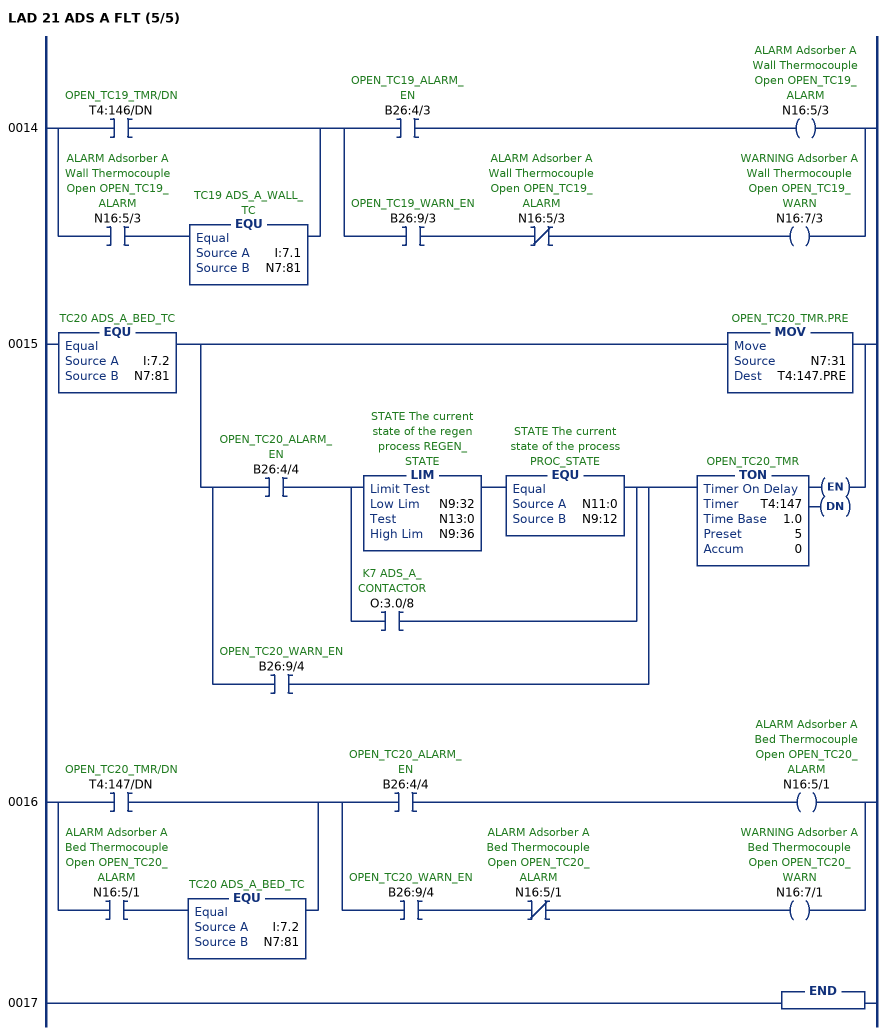
% Rung: 14 %
SOR BST XIC T4:146/DN NXB XIC N16:5/3 EQU I:7.1 N7:81 BND BST XIC B26:4/3 OTE N16:5/3 NXB XIC B26:9/3 XIO N16:5/3 OTE N16:7/3 BND EOR
%   T4:146  OPEN_TC19_TMR %
%   N16:5/3  OPEN_TC19_ALARM  "ALARM Adsorber A Wall Thermocouple Open" %
%   I:7.1  ADS_A_WALL_TC  "TC19" %
%   N7:81  TC_OPEN_SP  "CONFIG The value read by an open TC input" %
%   B26:4/3  OPEN_TC19_ALARM_EN %
%   B26:9/3  OPEN_TC19_WARN_EN %
%   N16:7/3  OPEN_TC19_WARN  "WARNING Adsorber A Wall Thermocouple Open" %
% Rung: 15 %
SOR EQU I:7.2 N7:81 BST MOV N7:31 T4:147.PRE NXB BST XIC B26:4/4 BST LIM N9:32 N13:0 N9:36 EQU N11:0 N9:12 NXB XIC O:3.0/8 BND NXB XIC B26:9/4 BND TON T4:147 1.0 5 0 BND EOR
%   I:7.2  ADS_A_BED_TC  "TC20" %
%   N7:81  TC_OPEN_SP  "CONFIG The value read by an open TC input" %
%   N7:31  OPEN_TC_DLY %
%   T4:147  OPEN_TC20_TMR %
%   B26:4/4  OPEN_TC20_ALARM_EN %
%   N9:32  REGEN_VENT  "STATE Regen Vent" %
%   N13:0  REGEN_STATE  "STATE The current state of the regen process" %
%   N9:36  REGEN_COOL  "STATE Regen Cool" %
%   N11:0  PROC_STATE  "STATE The current state of the process" %
%   N9:12  PROC_PFY_B_REG_A  "STATE Process Purify B" %
%   O:3.0/8  ADS_A_CONTACTOR  "K7" %
%   B26:9/4  OPEN_TC20_WARN_EN %
% Rung: 16 %
SOR BST XIC T4:147/DN NXB XIC N16:5/1 EQU I:7.2 N7:81 BND BST XIC B26:4/4 OTE N16:5/1 NXB XIC B26:9/4 XIO N16:5/1 OTE N16:7/1 BND EOR
%   T4:147  OPEN_TC20_TMR %
%   N16:5/1  OPEN_TC20_ALARM  "ALARM Adsorber A Bed Thermocouple Open" %
%   I:7.2  ADS_A_BED_TC  "TC20" %
%   N7:81  TC_OPEN_SP  "CONFIG The value read by an open TC input" %
%   B26:4/4  OPEN_TC20_ALARM_EN %
%   B26:9/4  OPEN_TC20_WARN_EN %
%   N16:7/1  OPEN_TC20_WARN  "WARNING Adsorber A Bed Thermocouple Open" %
% Rung: 17 %
SOR END EOR

LADDER 22 "ADS B"    % Controld Adsorber B %
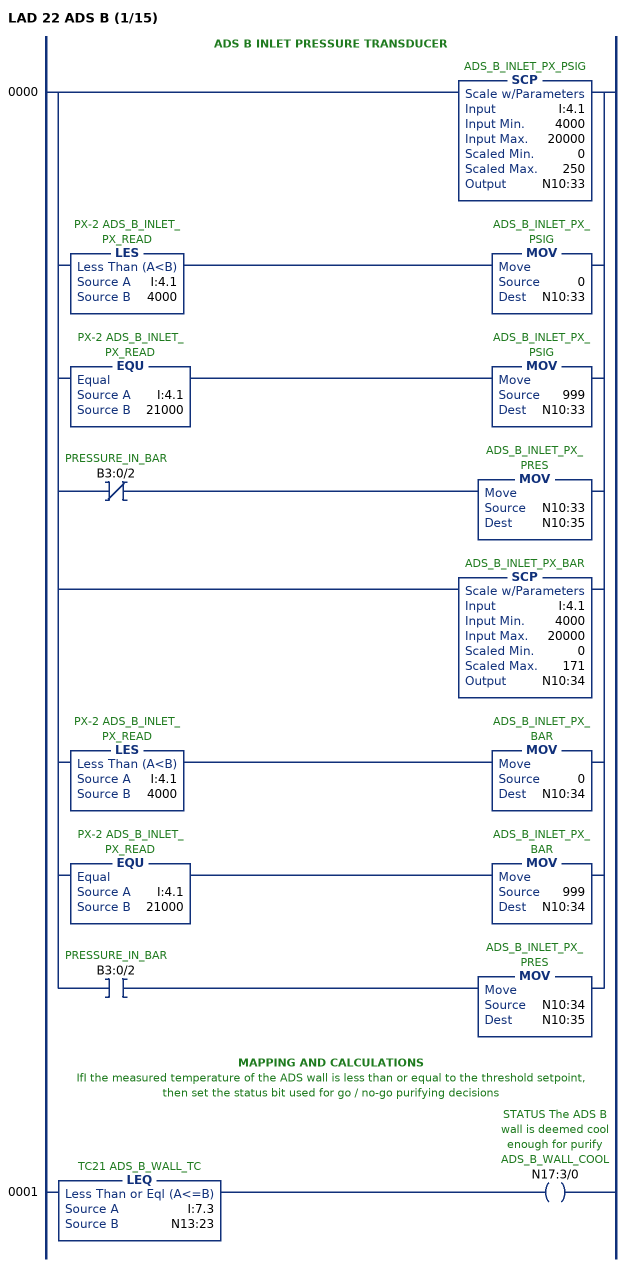
% Rung: 0 %
% TITLE: ADS B INLET PRESSURE TRANSDUCER %
SOR BST SCP I:4.1 4000 20000 0 250 N10:33 NXB LES I:4.1 4000 MOV 0 N10:33 NXB EQU I:4.1 21000 MOV 999 N10:33 NXB XIO B3:0/2 MOV N10:33 N10:35 NXB SCP I:4.1 4000 20000 0 171 N10:34 NXB LES I:4.1 4000 MOV 0 N10:34 NXB EQU I:4.1 21000 MOV 999 N10:34 NXB XIC B3:0/2 MOV N10:34 N10:35 BND EOR
%   I:4.1  ADS_B_INLET_PX_READ  "PX-2" %
%   N10:33  ADS_B_INLET_PX_PSIG %
%   B3:0/2  PRESSURE_IN_BAR %
%   N10:35  ADS_B_INLET_PX_PRES %
%   N10:34  ADS_B_INLET_PX_BAR %
% Rung: 1 %
% TITLE: MAPPING AND CALCULATIONS %
% IfI the measured temperature of the ADS wall is less than or equal to the threshold setpoint, then set the status bit used for go / no-go purifying decisions %
SOR LEQ I:7.3 N13:23 OTE N17:3/0 EOR
%   I:7.3  ADS_B_WALL_TC  "TC21" %
%   N13:23  ADS_WALL_TEMP_COOL  "CONFIG The temp at which the adsorber wall is deemed to be cool enough to purify" %
%   N17:3/0  ADS_B_WALL_COOL  "STATUS The ADS B wall is deemed cool enough for purify" %

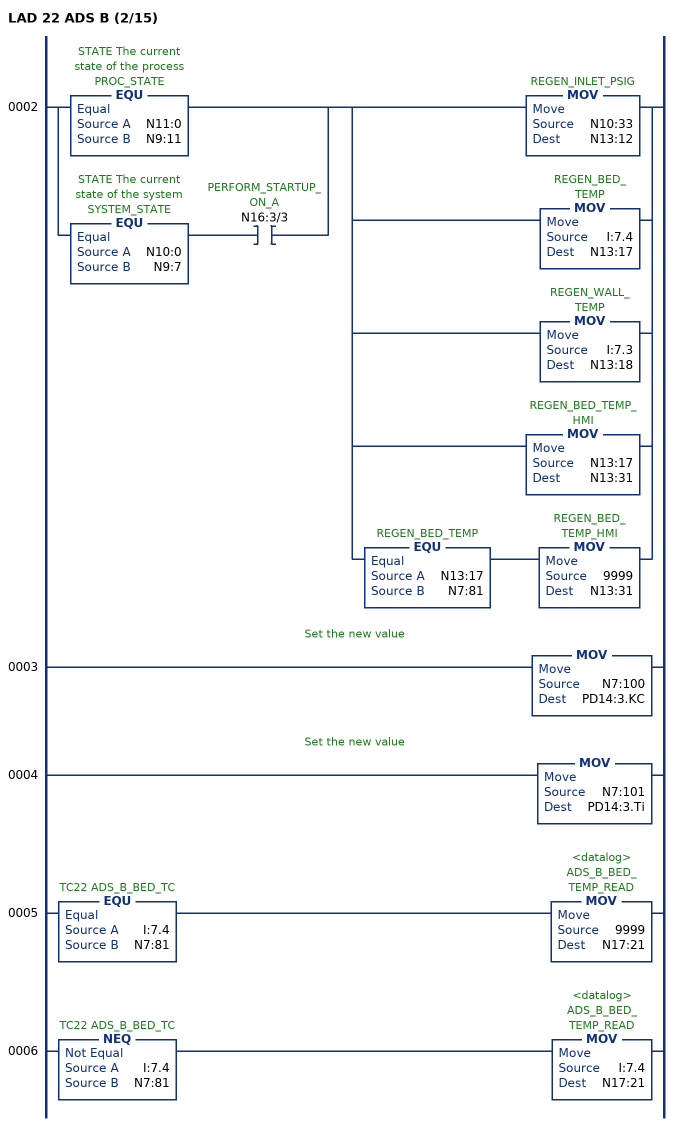
% Rung: 2 %
SOR BST EQU N11:0 N9:11 NXB EQU N10:0 N9:7 XIC N16:3/3 BND BST MOV N10:33 N13:12 NXB MOV I:7.4 N13:17 NXB MOV I:7.3 N13:18 NXB MOV N13:17 N13:31 NXB EQU N13:17 N7:81 MOV 9999 N13:31 BND EOR
%   N11:0  PROC_STATE  "STATE The current state of the process" %
%   N9:11  PROC_PFY_A_REG_B  "STATE Process Purify A" %
%   N10:0  SYSTEM_STATE  "STATE The current state of the system" %
%   N9:7  SYSTEM_COLD_START %
%   N16:3/3  PERFORM_STARTUP_ON_A %
%   N10:33  ADS_B_INLET_PX_PSIG %
%   N13:12  REGEN_INLET_PSIG %
%   I:7.4  ADS_B_BED_TC  "TC22" %
%   N13:17  REGEN_BED_TEMP %
%   I:7.3  ADS_B_WALL_TC  "TC21" %
%   N13:18  REGEN_WALL_TEMP %
%   N13:31  REGEN_BED_TEMP_HMI %
%   N7:81  TC_OPEN_SP  "CONFIG The value read by an open TC input" %
% Rung: 3 %
% Set the new value %
SOR MOV N7:100 PD14:3.KC EOR
%   N7:100  BLANKET_P  "CONFIG Blanket Proportional Gain New" %
% Rung: 4 %
% Set the new value %
SOR MOV N7:101 PD14:3.Ti EOR
%   N7:101  BLANKET_I  "CONFIG Blanket Integral Gain New" %
% Rung: 5 %
SOR EQU I:7.4 N7:81 MOV 9999 N17:21 EOR
%   I:7.4  ADS_B_BED_TC  "TC22" %
%   N7:81  TC_OPEN_SP  "CONFIG The value read by an open TC input" %
%   N17:21  ADS_B_BED_TEMP_READ  "<datalog>" %
% Rung: 6 %
SOR NEQ I:7.4 N7:81 MOV I:7.4 N17:21 EOR
%   I:7.4  ADS_B_BED_TC  "TC22" %
%   N7:81  TC_OPEN_SP  "CONFIG The value read by an open TC input" %
%   N17:21  ADS_B_BED_TEMP_READ  "<datalog>" %

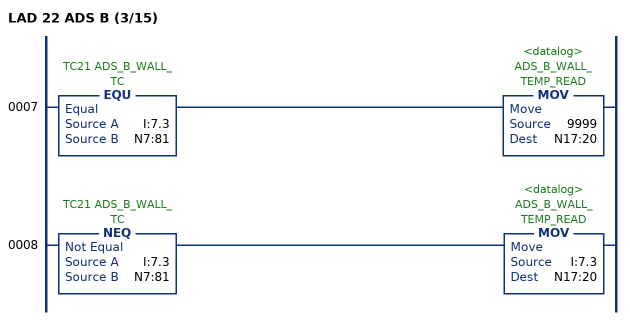
% Rung: 7 %
SOR EQU I:7.3 N7:81 MOV 9999 N17:20 EOR
%   I:7.3  ADS_B_WALL_TC  "TC21" %
%   N7:81  TC_OPEN_SP  "CONFIG The value read by an open TC input" %
%   N17:20  ADS_B_WALL_TEMP_READ  "<datalog>" %
% Rung: 8 %
SOR NEQ I:7.3 N7:81 MOV I:7.3 N17:20 EOR
%   I:7.3  ADS_B_WALL_TC  "TC21" %
%   N7:81  TC_OPEN_SP  "CONFIG The value read by an open TC input" %
%   N17:20  ADS_B_WALL_TEMP_READ  "<datalog>" %

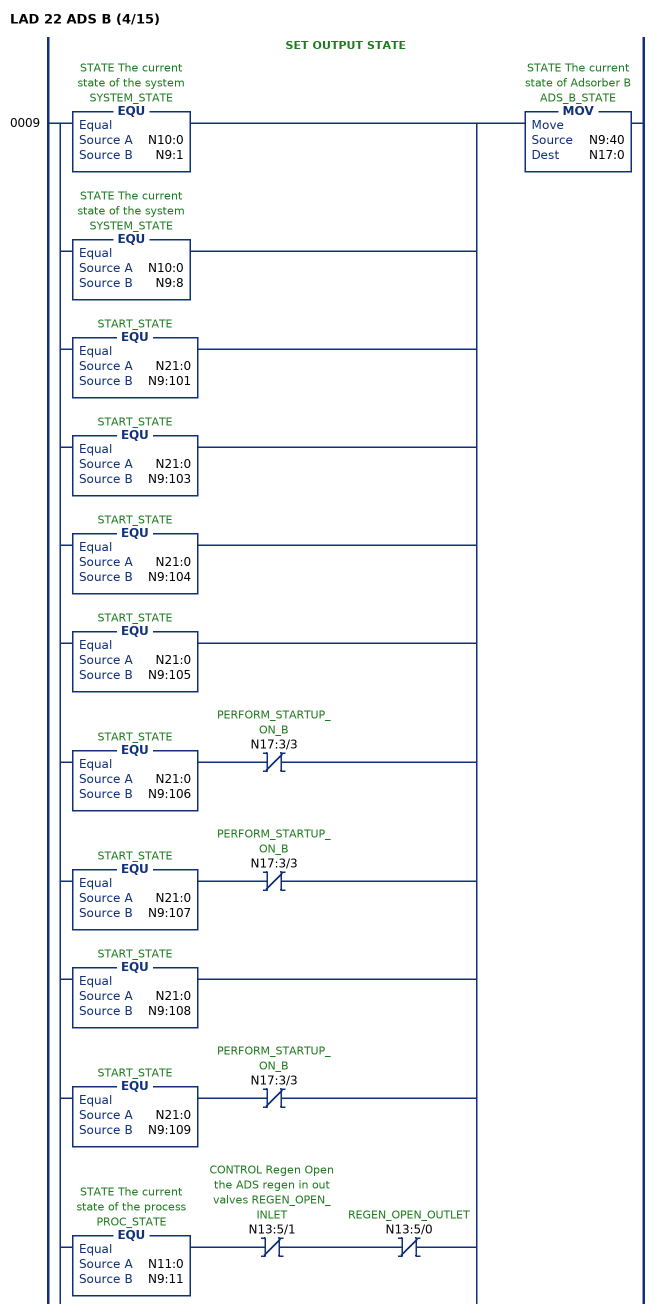

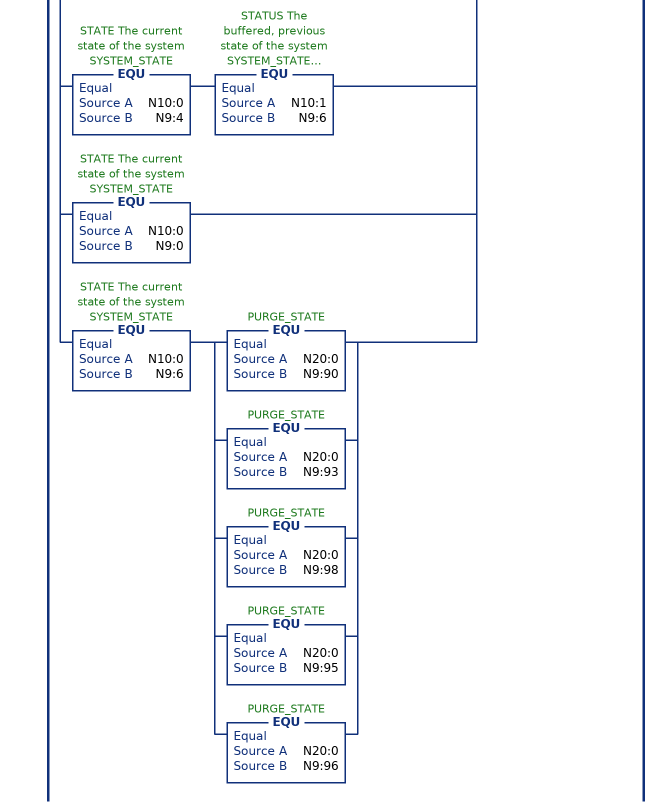
% Rung: 9 %
% TITLE: SET OUTPUT STATE %
SOR BST EQU N10:0 N9:1 NXB EQU N10:0 N9:8 NXB BST EQU N21:0 N9:101 NXB EQU N21:0 N9:103 NXB EQU N21:0 N9:104 NXB EQU N21:0 N9:105 NXB EQU N21:0 N9:106 XIO N17:3/3 NXB EQU N21:0 N9:107 XIO N17:3/3 NXB EQU N21:0 N9:108 NXB EQU N21:0 N9:109 XIO N17:3/3 BND NXB EQU N11:0 N9:11 XIO N13:5/1 XIO N13:5/0 NXB EQU N10:0 N9:4 EQU N10:1 N9:6 NXB EQU N10:0 N9:0 NXB EQU N10:0 N9:6 BST EQU N20:0 N9:90 NXB EQU N20:0 N9:93 NXB EQU N20:0 N9:98 NXB EQU N20:0 N9:95 NXB EQU N20:0 N9:96 BND BND MOV N9:40 N17:0 EOR
%   N10:0  SYSTEM_STATE  "STATE The current state of the system" %
%   N9:1  SYSTEM_STANDBY  "STATE System Process" %
%   N9:8  SYSTEM_SUPPLEMENTAL %
%   N21:0  START_STATE %
%   N9:101  START_COOL %
%   N9:103  START_VENT_GET_1 %
%   N9:104  START_HEAT %
%   N9:105  START_VENT_ALL %
%   N9:106  START_BACKFILL_1 %
%   N17:3/3  PERFORM_STARTUP_ON_B %
%   N9:107  START_VENT_ADS_2 %
%   N9:108  START_VENT_GET_2 %
%   N9:109  START_BACKFILL_2 %
%   N11:0  PROC_STATE  "STATE The current state of the process" %
%   N9:11  PROC_PFY_A_REG_B  "STATE Process Purify A" %
%   N13:5/1  REGEN_OPEN_INLET  "CONTROL Regen Open the ADS regen in out valves" %
%   N13:5/0  REGEN_OPEN_OUTLET %
%   N9:4  SYSTEM_ALARM  "STATE System Alarm" %
%   N10:1  SYSTEM_STATE_BUFFER  "STATUS The buffered, previous state of the system" %
%   N9:6  SYSTEM_PURGE %
%   N9:0  SYSTEM_OFFLINE %
%   N20:0  PURGE_STATE %
%   N9:90  PURGE_IDLE %
%   N9:93  PURGE_VENT_GETTER %
%   N9:98  PURGE_VENT_GET_2 %
%   N9:95  PURGE_FINAL_VENT %
%   N9:96  PURGE_DONE %
%   N9:40  ADS_STANDBY  "STATE ADS Standby" %
%   N17:0  ADS_B_STATE  "STATE The current state of Adsorber B" %

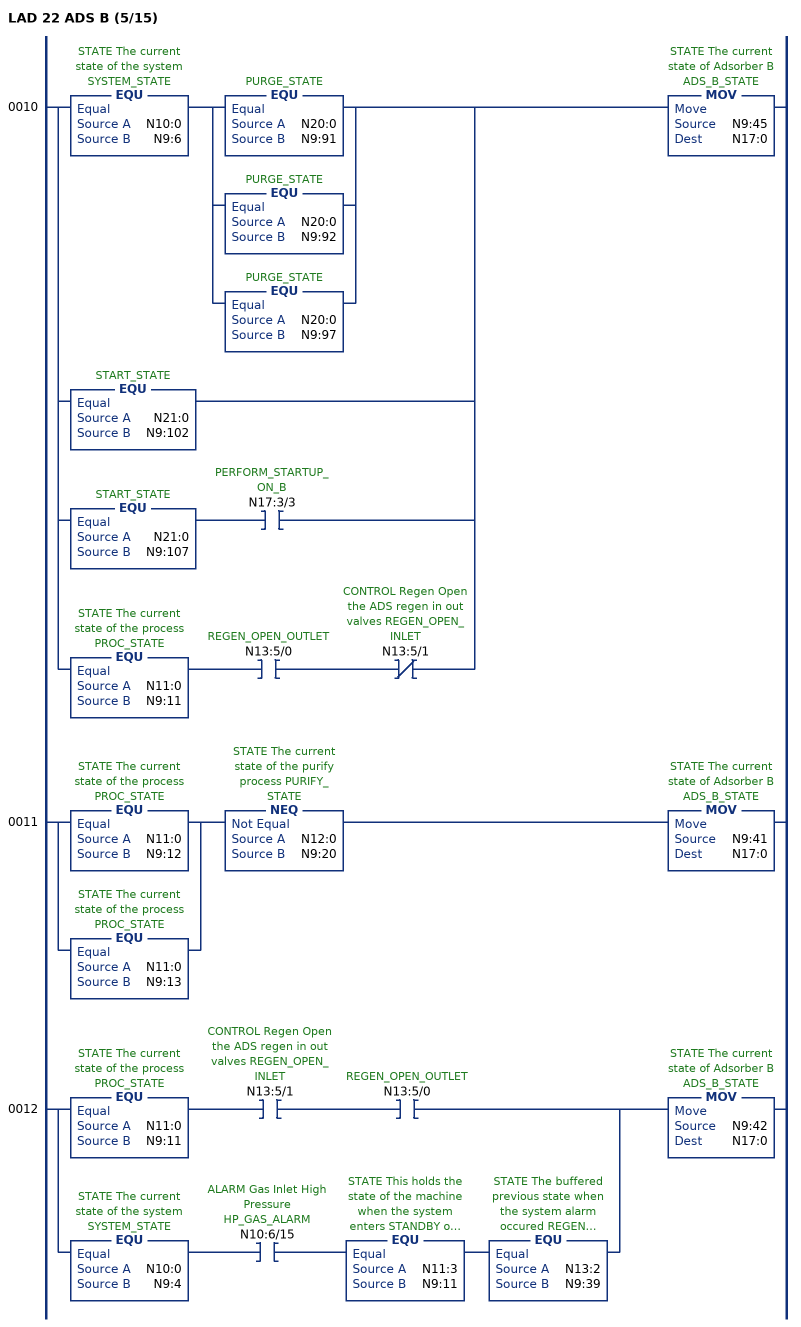
% Rung: 10 %
SOR BST EQU N10:0 N9:6 BST EQU N20:0 N9:91 NXB EQU N20:0 N9:92 NXB EQU N20:0 N9:97 BND NXB BST EQU N21:0 N9:102 NXB EQU N21:0 N9:107 XIC N17:3/3 BND NXB EQU N11:0 N9:11 XIC N13:5/0 XIO N13:5/1 BND MOV N9:45 N17:0 EOR
%   N10:0  SYSTEM_STATE  "STATE The current state of the system" %
%   N9:6  SYSTEM_PURGE %
%   N20:0  PURGE_STATE %
%   N9:91  PURGE_INIT_VENT %
%   N9:92  PURGE_VENT_ADSORBER %
%   N9:97  PURGE_VENT_ADS_2 %
%   N21:0  START_STATE %
%   N9:102  START_VENT_ADS_1 %
%   N9:107  START_VENT_ADS_2 %
%   N17:3/3  PERFORM_STARTUP_ON_B %
%   N11:0  PROC_STATE  "STATE The current state of the process" %
%   N9:11  PROC_PFY_A_REG_B  "STATE Process Purify A" %
%   N13:5/0  REGEN_OPEN_OUTLET %
%   N13:5/1  REGEN_OPEN_INLET  "CONTROL Regen Open the ADS regen in out valves" %
%   N9:45  ADS_VENT %
%   N17:0  ADS_B_STATE  "STATE The current state of Adsorber B" %
% Rung: 11 %
SOR BST EQU N11:0 N9:12 NXB EQU N11:0 N9:13 BND NEQ N12:0 N9:20 MOV N9:41 N17:0 EOR
%   N11:0  PROC_STATE  "STATE The current state of the process" %
%   N9:12  PROC_PFY_B_REG_A  "STATE Process Purify B" %
%   N9:13  PROC_OVERLAP  "STATE Process Purify Overlap" %
%   N12:0  PURIFY_STATE  "STATE The current state of the purify process" %
%   N9:20  PURIFY_STANDBY  "STATE Purify Standby" %
%   N9:41  ADS_PURIFY  "STATE ADS Purify" %
%   N17:0  ADS_B_STATE  "STATE The current state of Adsorber B" %
% Rung: 12 %
SOR BST EQU N11:0 N9:11 XIC N13:5/1 XIC N13:5/0 NXB EQU N10:0 N9:4 XIC N10:6/15 EQU N11:3 N9:11 EQU N13:2 N9:39 BND MOV N9:42 N17:0 EOR
%   N11:0  PROC_STATE  "STATE The current state of the process" %
%   N9:11  PROC_PFY_A_REG_B  "STATE Process Purify A" %
%   N13:5/1  REGEN_OPEN_INLET  "CONTROL Regen Open the ADS regen in out valves" %
%   N13:5/0  REGEN_OPEN_OUTLET %
%   N10:0  SYSTEM_STATE  "STATE The current state of the system" %
%   N9:4  SYSTEM_ALARM  "STATE System Alarm" %
%   N10:6/15  HP_GAS_ALARM  "ALARM Gas Inlet High Pressure" %
%   N11:3  PROC_STATE_BUFFER  "STATE This holds the state of the machine when the system enters STANDBY or ALARM" %
%   N13:2  REGEN_SYSTEM_BUFFER  "STATE The buffered previous state when the system alarm occured" %
%   N9:39  REGEN_BACKFILL %
%   N9:42  ADS_REGEN  "STATE ADS Regen" %
%   N17:0  ADS_B_STATE  "STATE The current state of Adsorber B" %

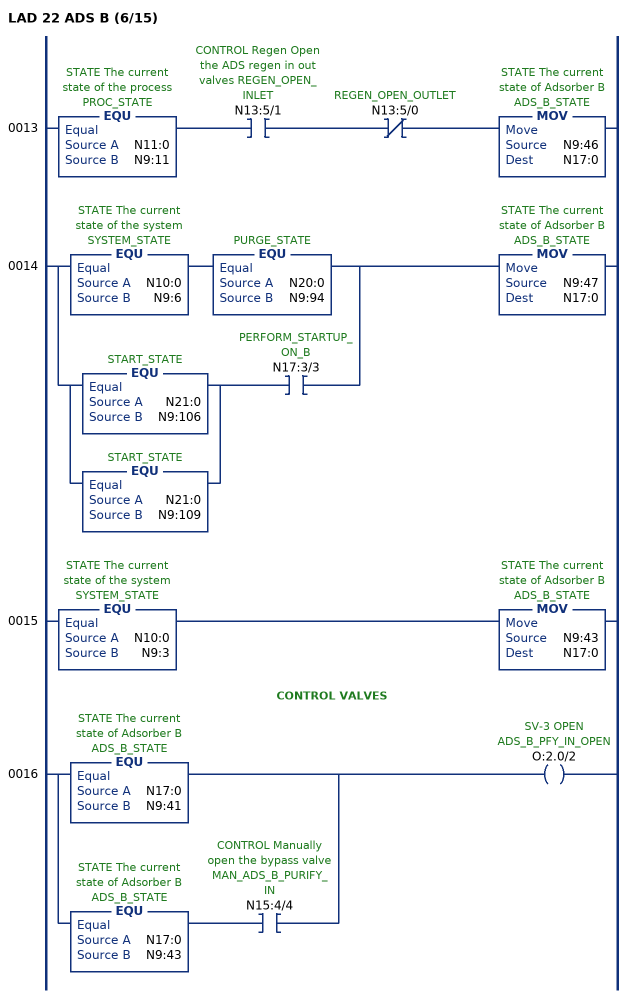
% Rung: 13 %
SOR EQU N11:0 N9:11 XIC N13:5/1 XIO N13:5/0 MOV N9:46 N17:0 EOR
%   N11:0  PROC_STATE  "STATE The current state of the process" %
%   N9:11  PROC_PFY_A_REG_B  "STATE Process Purify A" %
%   N13:5/1  REGEN_OPEN_INLET  "CONTROL Regen Open the ADS regen in out valves" %
%   N13:5/0  REGEN_OPEN_OUTLET %
%   N9:46  ADS_REGEN_BACKFILL %
%   N17:0  ADS_B_STATE  "STATE The current state of Adsorber B" %
% Rung: 14 %
SOR BST EQU N10:0 N9:6 EQU N20:0 N9:94 NXB BST EQU N21:0 N9:106 NXB EQU N21:0 N9:109 BND XIC N17:3/3 BND MOV N9:47 N17:0 EOR
%   N10:0  SYSTEM_STATE  "STATE The current state of the system" %
%   N9:6  SYSTEM_PURGE %
%   N20:0  PURGE_STATE %
%   N9:94  PURGE_BACKFILL %
%   N21:0  START_STATE %
%   N9:106  START_BACKFILL_1 %
%   N9:109  START_BACKFILL_2 %
%   N17:3/3  PERFORM_STARTUP_ON_B %
%   N9:47  ADS_BACKFILL %
%   N17:0  ADS_B_STATE  "STATE The current state of Adsorber B" %
% Rung: 15 %
SOR EQU N10:0 N9:3 MOV N9:43 N17:0 EOR
%   N10:0  SYSTEM_STATE  "STATE The current state of the system" %
%   N9:3  SYSTEM_MANUAL  "STATE System Manual" %
%   N9:43  ADS_MANUAL  "STATE ADS Manual" %
%   N17:0  ADS_B_STATE  "STATE The current state of Adsorber B" %
% Rung: 16 %
% TITLE: CONTROL VALVES %
SOR BST EQU N17:0 N9:41 NXB EQU N17:0 N9:43 XIC N15:4/4 BND OTE O:2.0/2 EOR
%   N17:0  ADS_B_STATE  "STATE The current state of Adsorber B" %
%   N9:41  ADS_PURIFY  "STATE ADS Purify" %
%   N9:43  ADS_MANUAL  "STATE ADS Manual" %
%   N15:4/4  MAN_ADS_B_PURIFY_IN  "CONTROL Manually open the bypass valve" %
%   O:2.0/2  ADS_B_PFY_IN_OPEN  "SV-3 OPEN" %

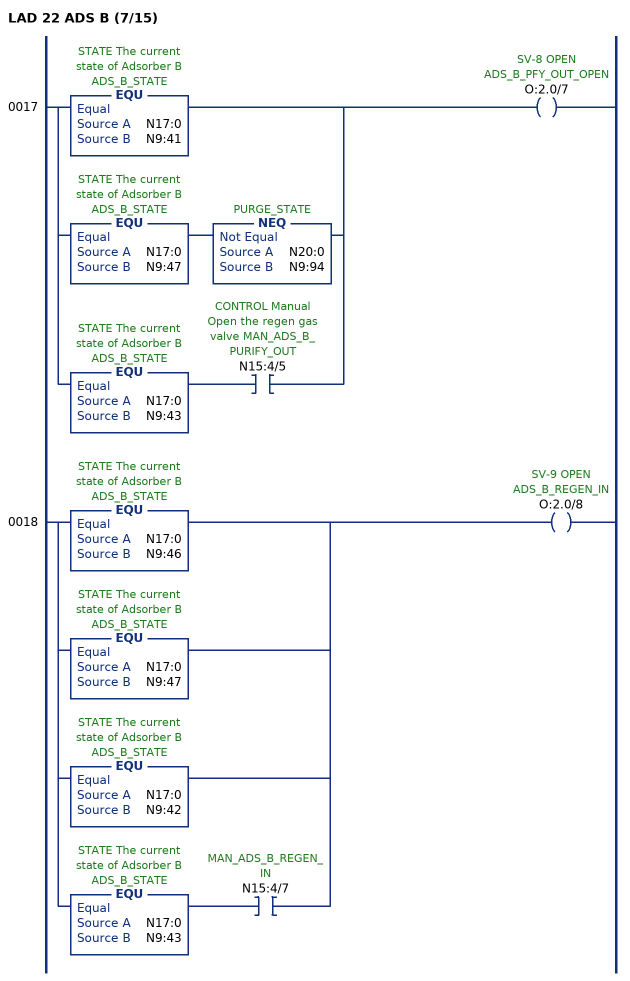
% Rung: 17 %
SOR BST EQU N17:0 N9:41 NXB EQU N17:0 N9:47 NEQ N20:0 N9:94 NXB EQU N17:0 N9:43 XIC N15:4/5 BND OTE O:2.0/7 EOR
%   N17:0  ADS_B_STATE  "STATE The current state of Adsorber B" %
%   N9:41  ADS_PURIFY  "STATE ADS Purify" %
%   N9:47  ADS_BACKFILL %
%   N20:0  PURGE_STATE %
%   N9:94  PURGE_BACKFILL %
%   N9:43  ADS_MANUAL  "STATE ADS Manual" %
%   N15:4/5  MAN_ADS_B_PURIFY_OUT  "CONTROL Manual Open the regen gas valve" %
%   O:2.0/7  ADS_B_PFY_OUT_OPEN  "SV-8 OPEN" %
% Rung: 18 %
SOR BST EQU N17:0 N9:46 NXB EQU N17:0 N9:47 NXB EQU N17:0 N9:42 NXB EQU N17:0 N9:43 XIC N15:4/7 BND OTE O:2.0/8 EOR
%   N17:0  ADS_B_STATE  "STATE The current state of Adsorber B" %
%   N9:46  ADS_REGEN_BACKFILL %
%   N9:47  ADS_BACKFILL %
%   N9:42  ADS_REGEN  "STATE ADS Regen" %
%   N9:43  ADS_MANUAL  "STATE ADS Manual" %
%   N15:4/7  MAN_ADS_B_REGEN_IN %
%   O:2.0/8  ADS_B_REGEN_IN  "SV-9 OPEN" %

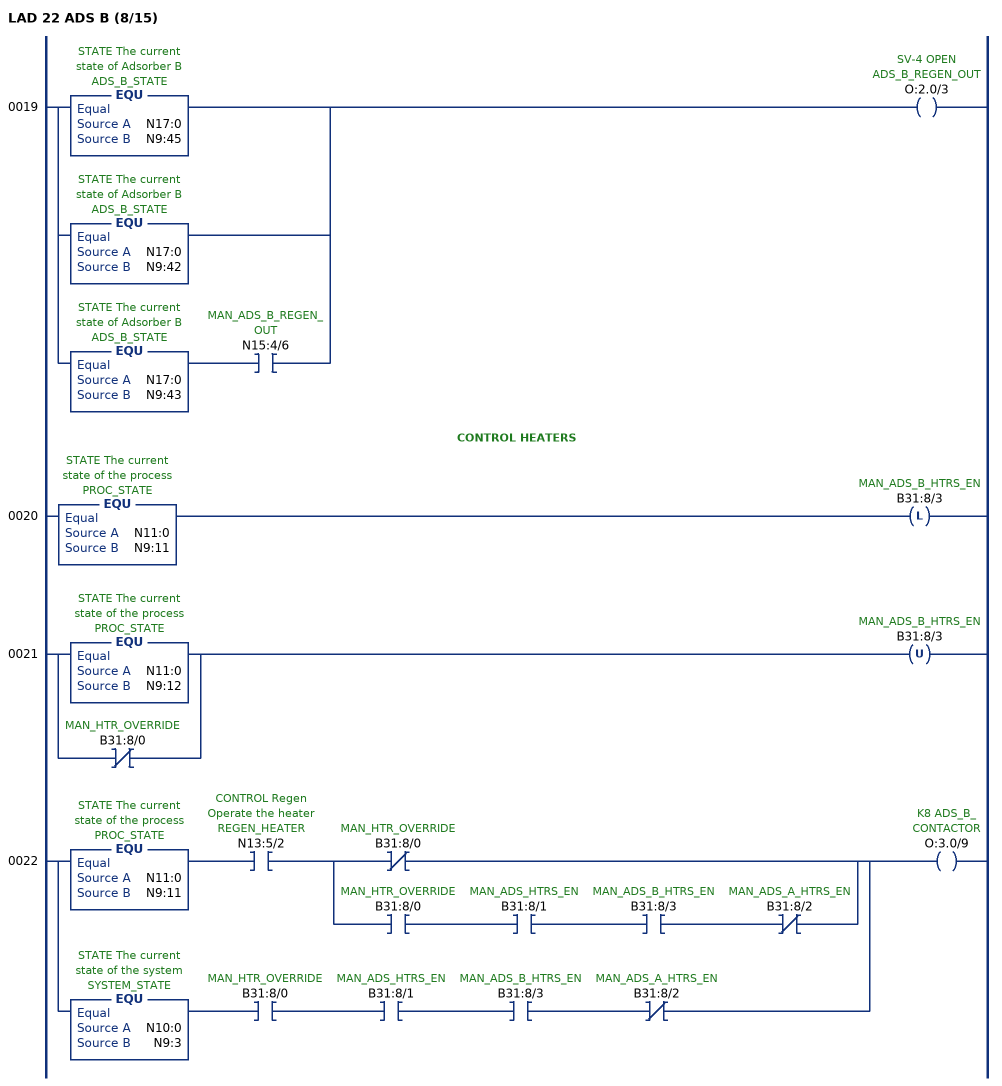
% Rung: 19 %
SOR BST EQU N17:0 N9:45 NXB EQU N17:0 N9:42 NXB EQU N17:0 N9:43 XIC N15:4/6 BND OTE O:2.0/3 EOR
%   N17:0  ADS_B_STATE  "STATE The current state of Adsorber B" %
%   N9:45  ADS_VENT %
%   N9:42  ADS_REGEN  "STATE ADS Regen" %
%   N9:43  ADS_MANUAL  "STATE ADS Manual" %
%   N15:4/6  MAN_ADS_B_REGEN_OUT %
%   O:2.0/3  ADS_B_REGEN_OUT  "SV-4 OPEN" %
% Rung: 20 %
% TITLE: CONTROL HEATERS %
SOR EQU N11:0 N9:11 OTL B31:8/3 EOR
%   N11:0  PROC_STATE  "STATE The current state of the process" %
%   N9:11  PROC_PFY_A_REG_B  "STATE Process Purify A" %
%   B31:8/3  MAN_ADS_B_HTRS_EN %
% Rung: 21 %
SOR BST EQU N11:0 N9:12 NXB XIO B31:8/0 BND OTU B31:8/3 EOR
%   N11:0  PROC_STATE  "STATE The current state of the process" %
%   N9:12  PROC_PFY_B_REG_A  "STATE Process Purify B" %
%   B31:8/0  MAN_HTR_OVERRIDE %
%   B31:8/3  MAN_ADS_B_HTRS_EN %
% Rung: 22 %
SOR BST EQU N11:0 N9:11 XIC N13:5/2 BST XIO B31:8/0 NXB XIC B31:8/0 XIC B31:8/1 XIC B31:8/3 XIO B31:8/2 BND NXB EQU N10:0 N9:3 XIC B31:8/0 XIC B31:8/1 XIC B31:8/3 XIO B31:8/2 BND OTE O:3.0/9 EOR
%   N11:0  PROC_STATE  "STATE The current state of the process" %
%   N9:11  PROC_PFY_A_REG_B  "STATE Process Purify A" %
%   N13:5/2  REGEN_HEATER  "CONTROL Regen Operate the heater" %
%   B31:8/0  MAN_HTR_OVERRIDE %
%   B31:8/1  MAN_ADS_HTRS_EN %
%   B31:8/3  MAN_ADS_B_HTRS_EN %
%   B31:8/2  MAN_ADS_A_HTRS_EN %
%   N10:0  SYSTEM_STATE  "STATE The current state of the system" %
%   N9:3  SYSTEM_MANUAL  "STATE System Manual" %
%   O:3.0/9  ADS_B_CONTACTOR  "K8" %

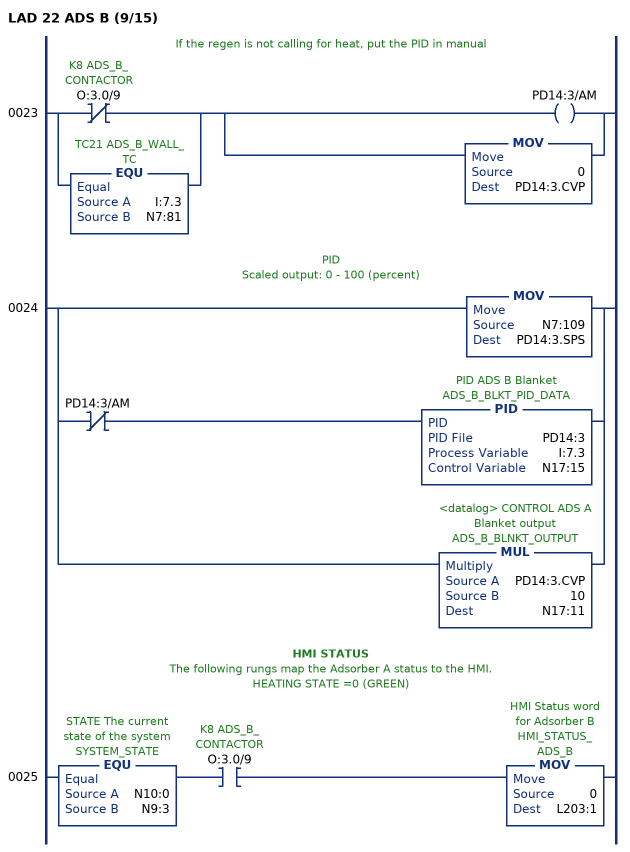
% Rung: 23 %
% If the regen is not calling for heat, put the PID in manual %
SOR BST XIO O:3.0/9 NXB EQU I:7.3 N7:81 BND BST OTE PD14:3/AM NXB MOV 0 PD14:3.CVP BND EOR
%   O:3.0/9  ADS_B_CONTACTOR  "K8" %
%   I:7.3  ADS_B_WALL_TC  "TC21" %
%   N7:81  TC_OPEN_SP  "CONFIG The value read by an open TC input" %
% Rung: 24 %
% PID
% Scaled output: 0 - 100 (percent) %
SOR BST MOV N7:109 PD14:3.SPS NXB XIO PD14:3/AM PID PD14:3 I:7.3 N17:15 NXB MUL PD14:3.CVP 10 N17:11 BND EOR
%   N7:109  BLANKET_SP  "<datalog> CONTROL Blanket PID Setpoint" %
%   PD14:3  ADS_B_BLKT_PID_DATA  "PID ADS B Blanket" %
%   I:7.3  ADS_B_WALL_TC  "TC21" %
%   N17:15  ADS_B_BLKT_OUTPT_RAW  "CONTROL ADS B Blanket PID Output Raw" %
%   N17:11  ADS_B_BLNKT_OUTPUT  "<datalog> CONTROL ADS A Blanket output" %
% Rung: 25 %
% TITLE: HMI STATUS %
% The following rungs map the Adsorber A status to the HMI.
% HEATING STATE =0 (GREEN) %
SOR EQU N10:0 N9:3 XIC O:3.0/9 MOV 0 L203:1 EOR
%   N10:0  SYSTEM_STATE  "STATE The current state of the system" %
%   N9:3  SYSTEM_MANUAL  "STATE System Manual" %
%   O:3.0/9  ADS_B_CONTACTOR  "K8" %
%   L203:1  HMI_STATUS_ADS_B  "HMI Status word for Adsorber B" %

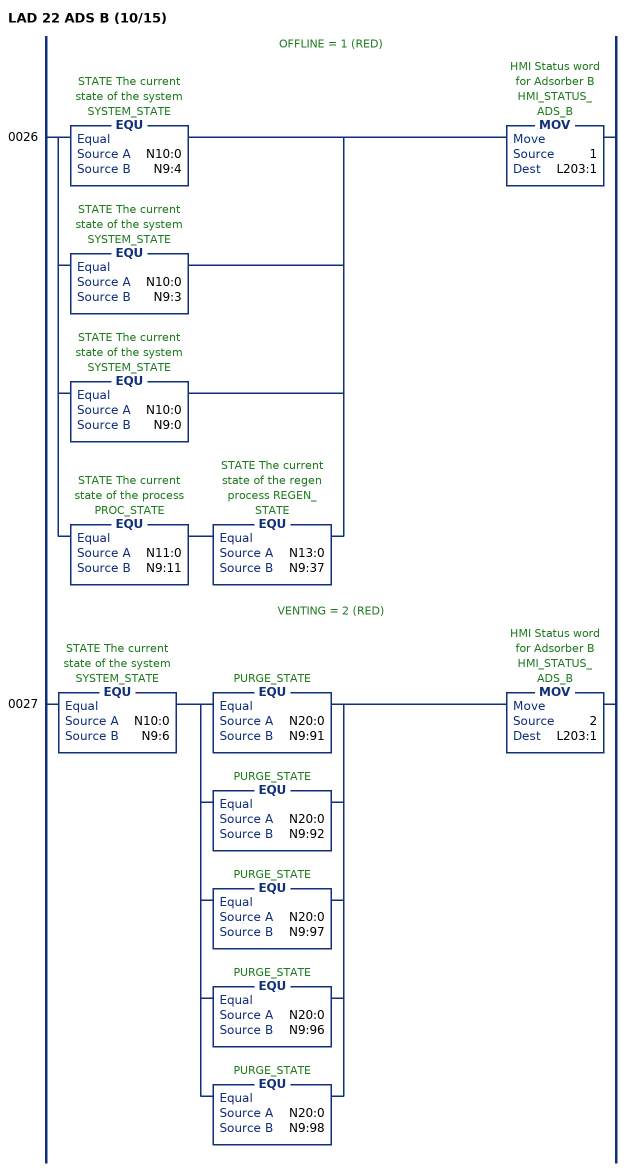
% Rung: 26 %
% OFFLINE = 1 (RED) %
SOR BST BST EQU N10:0 N9:4 NXB EQU N10:0 N9:3 NXB EQU N10:0 N9:0 BND NXB EQU N11:0 N9:11 EQU N13:0 N9:37 BND MOV 1 L203:1 EOR
%   N10:0  SYSTEM_STATE  "STATE The current state of the system" %
%   N9:4  SYSTEM_ALARM  "STATE System Alarm" %
%   N9:3  SYSTEM_MANUAL  "STATE System Manual" %
%   N9:0  SYSTEM_OFFLINE %
%   N11:0  PROC_STATE  "STATE The current state of the process" %
%   N9:11  PROC_PFY_A_REG_B  "STATE Process Purify A" %
%   N13:0  REGEN_STATE  "STATE The current state of the regen process" %
%   N9:37  REGEN_ALARM  "STATE Regen Alarm" %
%   L203:1  HMI_STATUS_ADS_B  "HMI Status word for Adsorber B" %
% Rung: 27 %
% VENTING = 2 (RED) %
SOR EQU N10:0 N9:6 BST EQU N20:0 N9:91 NXB EQU N20:0 N9:92 NXB EQU N20:0 N9:97 NXB EQU N20:0 N9:96 NXB EQU N20:0 N9:98 BND MOV 2 L203:1 EOR
%   N10:0  SYSTEM_STATE  "STATE The current state of the system" %
%   N9:6  SYSTEM_PURGE %
%   N20:0  PURGE_STATE %
%   N9:91  PURGE_INIT_VENT %
%   N9:92  PURGE_VENT_ADSORBER %
%   N9:97  PURGE_VENT_ADS_2 %
%   N9:96  PURGE_DONE %
%   N9:98  PURGE_VENT_GET_2 %
%   L203:1  HMI_STATUS_ADS_B  "HMI Status word for Adsorber B" %

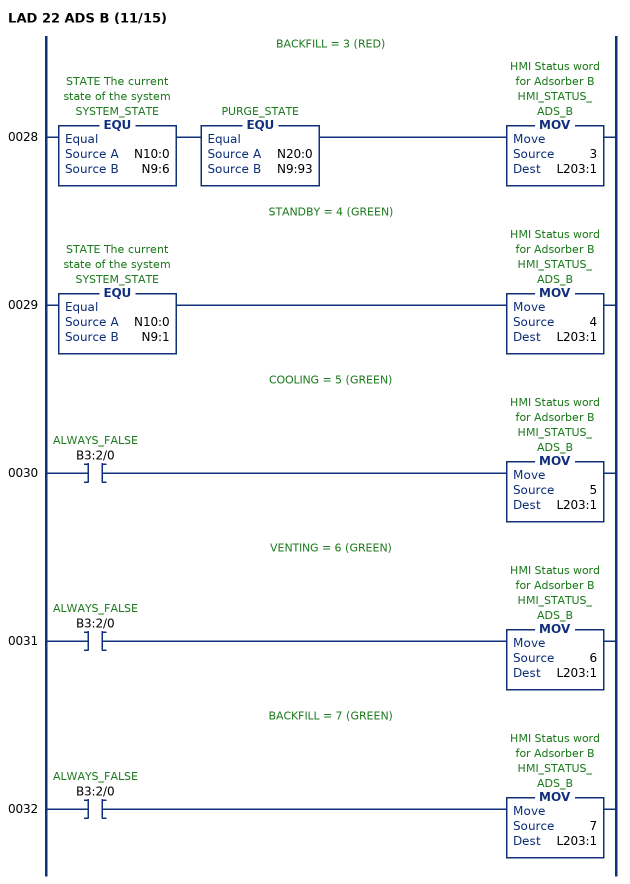
% Rung: 28 %
% BACKFILL = 3 (RED) %
SOR EQU N10:0 N9:6 EQU N20:0 N9:93 MOV 3 L203:1 EOR
%   N10:0  SYSTEM_STATE  "STATE The current state of the system" %
%   N9:6  SYSTEM_PURGE %
%   N20:0  PURGE_STATE %
%   N9:93  PURGE_VENT_GETTER %
%   L203:1  HMI_STATUS_ADS_B  "HMI Status word for Adsorber B" %
% Rung: 29 %
% STANDBY = 4 (GREEN) %
SOR EQU N10:0 N9:1 MOV 4 L203:1 EOR
%   N10:0  SYSTEM_STATE  "STATE The current state of the system" %
%   N9:1  SYSTEM_STANDBY  "STATE System Process" %
%   L203:1  HMI_STATUS_ADS_B  "HMI Status word for Adsorber B" %
% Rung: 30 %
% COOLING = 5 (GREEN) %
SOR XIC B3:2/0 MOV 5 L203:1 EOR
%   B3:2/0  ALWAYS_FALSE %
%   L203:1  HMI_STATUS_ADS_B  "HMI Status word for Adsorber B" %
% Rung: 31 %
% VENTING = 6 (GREEN) %
SOR XIC B3:2/0 MOV 6 L203:1 EOR
%   B3:2/0  ALWAYS_FALSE %
%   L203:1  HMI_STATUS_ADS_B  "HMI Status word for Adsorber B" %
% Rung: 32 %
% BACKFILL = 7 (GREEN) %
SOR XIC B3:2/0 MOV 7 L203:1 EOR
%   B3:2/0  ALWAYS_FALSE %
%   L203:1  HMI_STATUS_ADS_B  "HMI Status word for Adsorber B" %

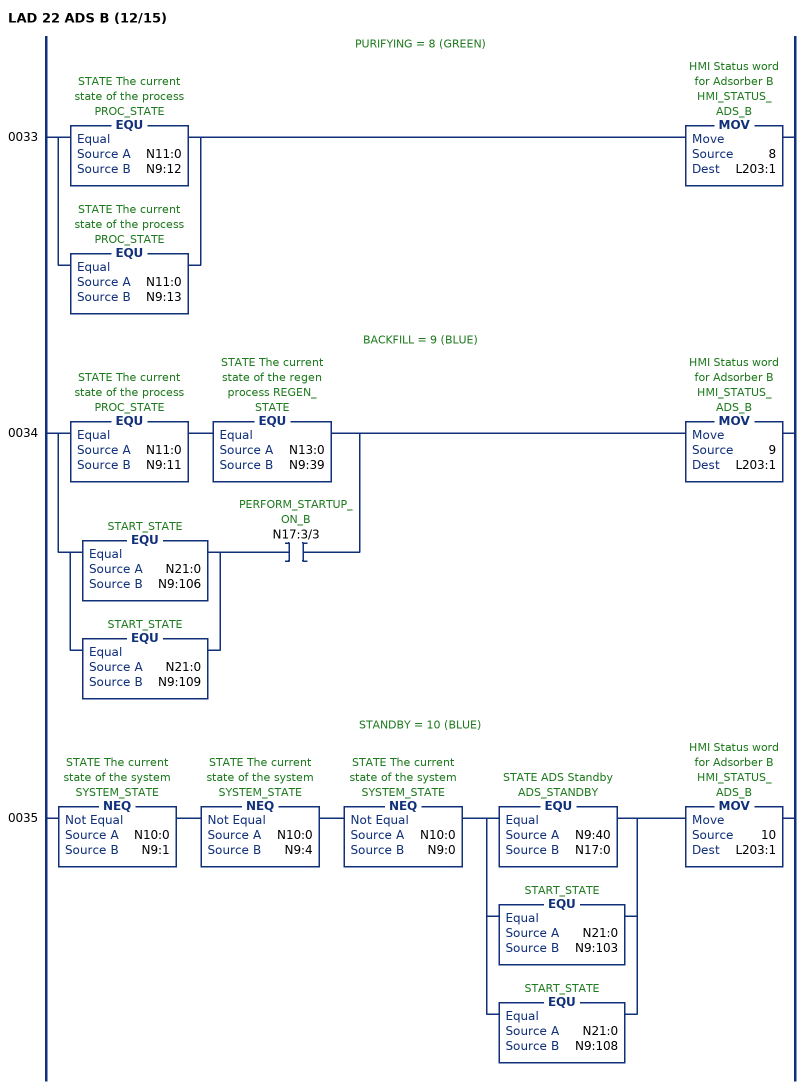
% Rung: 33 %
% PURIFYING = 8 (GREEN) %
SOR BST EQU N11:0 N9:12 NXB EQU N11:0 N9:13 BND MOV 8 L203:1 EOR
%   N11:0  PROC_STATE  "STATE The current state of the process" %
%   N9:12  PROC_PFY_B_REG_A  "STATE Process Purify B" %
%   N9:13  PROC_OVERLAP  "STATE Process Purify Overlap" %
%   L203:1  HMI_STATUS_ADS_B  "HMI Status word for Adsorber B" %
% Rung: 34 %
% BACKFILL = 9 (BLUE) %
SOR BST EQU N11:0 N9:11 EQU N13:0 N9:39 NXB BST EQU N21:0 N9:106 NXB EQU N21:0 N9:109 BND XIC N17:3/3 BND MOV 9 L203:1 EOR
%   N11:0  PROC_STATE  "STATE The current state of the process" %
%   N9:11  PROC_PFY_A_REG_B  "STATE Process Purify A" %
%   N13:0  REGEN_STATE  "STATE The current state of the regen process" %
%   N9:39  REGEN_BACKFILL %
%   N21:0  START_STATE %
%   N9:106  START_BACKFILL_1 %
%   N9:109  START_BACKFILL_2 %
%   N17:3/3  PERFORM_STARTUP_ON_B %
%   L203:1  HMI_STATUS_ADS_B  "HMI Status word for Adsorber B" %
% Rung: 35 %
% STANDBY = 10 (BLUE) %
SOR NEQ N10:0 N9:1 NEQ N10:0 N9:4 NEQ N10:0 N9:0 BST EQU N9:40 N17:0 NXB EQU N21:0 N9:103 NXB EQU N21:0 N9:108 BND MOV 10 L203:1 EOR
%   N10:0  SYSTEM_STATE  "STATE The current state of the system" %
%   N9:1  SYSTEM_STANDBY  "STATE System Process" %
%   N9:4  SYSTEM_ALARM  "STATE System Alarm" %
%   N9:0  SYSTEM_OFFLINE %
%   N9:40  ADS_STANDBY  "STATE ADS Standby" %
%   N17:0  ADS_B_STATE  "STATE The current state of Adsorber B" %
%   N21:0  START_STATE %
%   N9:103  START_VENT_GET_1 %
%   N9:108  START_VENT_GET_2 %
%   L203:1  HMI_STATUS_ADS_B  "HMI Status word for Adsorber B" %

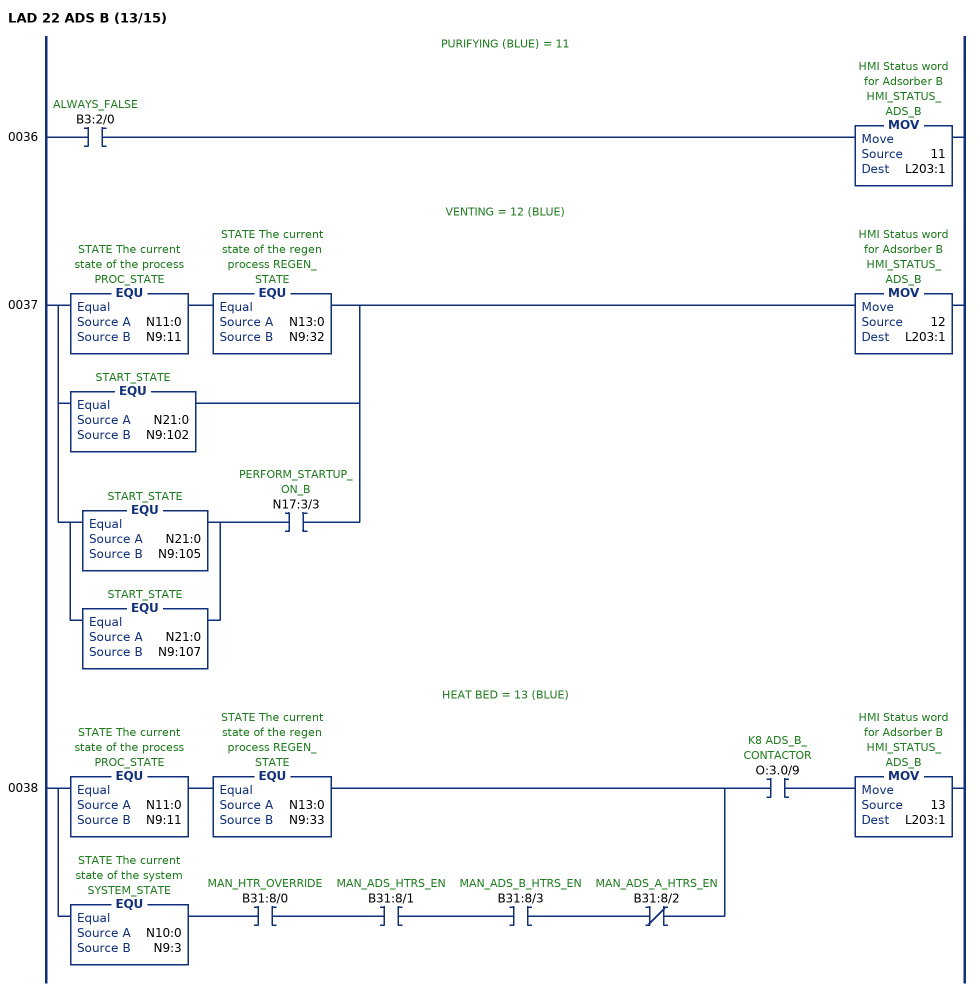
% Rung: 36 %
% PURIFYING (BLUE) = 11 %
SOR XIC B3:2/0 MOV 11 L203:1 EOR
%   B3:2/0  ALWAYS_FALSE %
%   L203:1  HMI_STATUS_ADS_B  "HMI Status word for Adsorber B" %
% Rung: 37 %
% VENTING = 12 (BLUE) %
SOR BST EQU N11:0 N9:11 EQU N13:0 N9:32 NXB BST EQU N21:0 N9:102 NXB BST EQU N21:0 N9:105 NXB EQU N21:0 N9:107 BND XIC N17:3/3 BND BND MOV 12 L203:1 EOR
%   N11:0  PROC_STATE  "STATE The current state of the process" %
%   N9:11  PROC_PFY_A_REG_B  "STATE Process Purify A" %
%   N13:0  REGEN_STATE  "STATE The current state of the regen process" %
%   N9:32  REGEN_VENT  "STATE Regen Vent" %
%   N21:0  START_STATE %
%   N9:102  START_VENT_ADS_1 %
%   N9:105  START_VENT_ALL %
%   N9:107  START_VENT_ADS_2 %
%   N17:3/3  PERFORM_STARTUP_ON_B %
%   L203:1  HMI_STATUS_ADS_B  "HMI Status word for Adsorber B" %
% Rung: 38 %
% HEAT BED = 13 (BLUE) %
SOR BST EQU N11:0 N9:11 EQU N13:0 N9:33 NXB EQU N10:0 N9:3 XIC B31:8/0 XIC B31:8/1 XIC B31:8/3 XIO B31:8/2 BND XIC O:3.0/9 MOV 13 L203:1 EOR
%   N11:0  PROC_STATE  "STATE The current state of the process" %
%   N9:11  PROC_PFY_A_REG_B  "STATE Process Purify A" %
%   N13:0  REGEN_STATE  "STATE The current state of the regen process" %
%   N9:33  REGEN_HEAT_BED  "STATE Regen Heat wall" %
%   N10:0  SYSTEM_STATE  "STATE The current state of the system" %
%   N9:3  SYSTEM_MANUAL  "STATE System Manual" %
%   B31:8/0  MAN_HTR_OVERRIDE %
%   B31:8/1  MAN_ADS_HTRS_EN %
%   B31:8/3  MAN_ADS_B_HTRS_EN %
%   B31:8/2  MAN_ADS_A_HTRS_EN %
%   O:3.0/9  ADS_B_CONTACTOR  "K8" %
%   L203:1  HMI_STATUS_ADS_B  "HMI Status word for Adsorber B" %

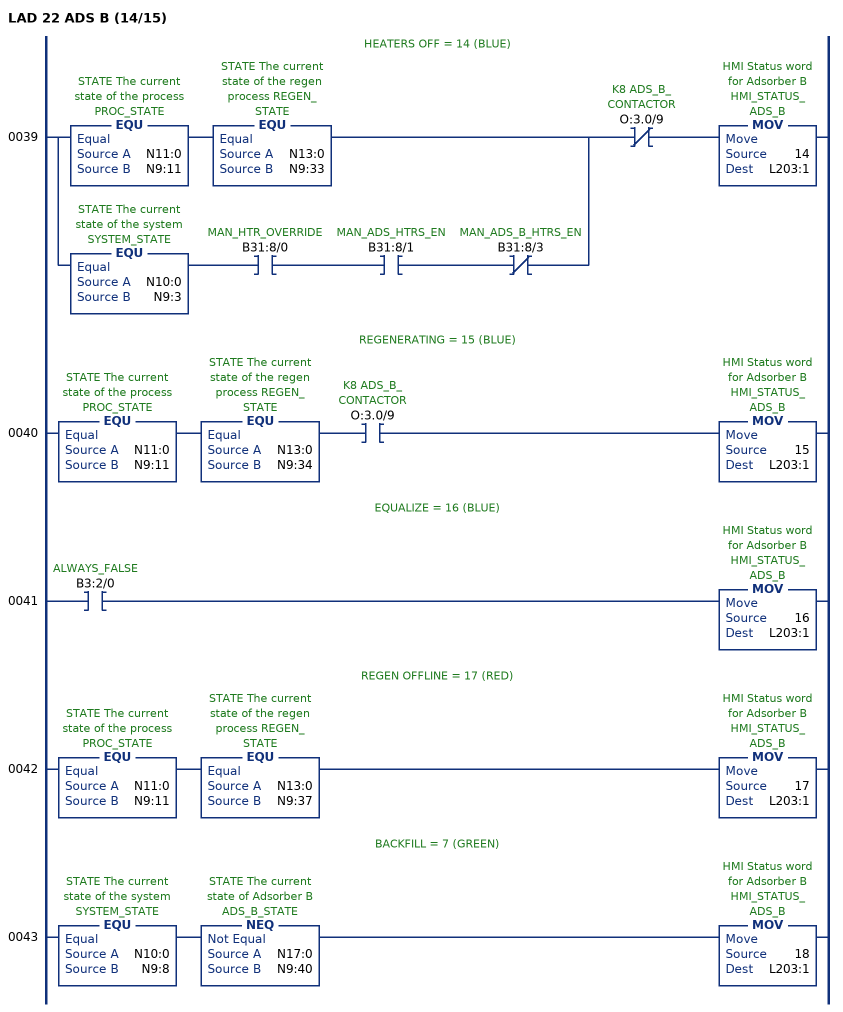
% Rung: 39 %
% HEATERS OFF = 14 (BLUE) %
SOR BST EQU N11:0 N9:11 EQU N13:0 N9:33 NXB EQU N10:0 N9:3 XIC B31:8/0 XIC B31:8/1 XIO B31:8/3 BND XIO O:3.0/9 MOV 14 L203:1 EOR
%   N11:0  PROC_STATE  "STATE The current state of the process" %
%   N9:11  PROC_PFY_A_REG_B  "STATE Process Purify A" %
%   N13:0  REGEN_STATE  "STATE The current state of the regen process" %
%   N9:33  REGEN_HEAT_BED  "STATE Regen Heat wall" %
%   N10:0  SYSTEM_STATE  "STATE The current state of the system" %
%   N9:3  SYSTEM_MANUAL  "STATE System Manual" %
%   B31:8/0  MAN_HTR_OVERRIDE %
%   B31:8/1  MAN_ADS_HTRS_EN %
%   B31:8/3  MAN_ADS_B_HTRS_EN %
%   O:3.0/9  ADS_B_CONTACTOR  "K8" %
%   L203:1  HMI_STATUS_ADS_B  "HMI Status word for Adsorber B" %
% Rung: 40 %
% REGENERATING = 15 (BLUE) %
SOR EQU N11:0 N9:11 EQU N13:0 N9:34 XIC O:3.0/9 MOV 15 L203:1 EOR
%   N11:0  PROC_STATE  "STATE The current state of the process" %
%   N9:11  PROC_PFY_A_REG_B  "STATE Process Purify A" %
%   N13:0  REGEN_STATE  "STATE The current state of the regen process" %
%   N9:34  REGEN_RUN  "STATE Regen Running" %
%   O:3.0/9  ADS_B_CONTACTOR  "K8" %
%   L203:1  HMI_STATUS_ADS_B  "HMI Status word for Adsorber B" %
% Rung: 41 %
% EQUALIZE = 16 (BLUE) %
SOR XIC B3:2/0 MOV 16 L203:1 EOR
%   B3:2/0  ALWAYS_FALSE %
%   L203:1  HMI_STATUS_ADS_B  "HMI Status word for Adsorber B" %
% Rung: 42 %
% REGEN OFFLINE = 17 (RED) %
SOR EQU N11:0 N9:11 EQU N13:0 N9:37 MOV 17 L203:1 EOR
%   N11:0  PROC_STATE  "STATE The current state of the process" %
%   N9:11  PROC_PFY_A_REG_B  "STATE Process Purify A" %
%   N13:0  REGEN_STATE  "STATE The current state of the regen process" %
%   N9:37  REGEN_ALARM  "STATE Regen Alarm" %
%   L203:1  HMI_STATUS_ADS_B  "HMI Status word for Adsorber B" %
% Rung: 43 %
% BACKFILL = 7 (GREEN) %
SOR EQU N10:0 N9:8 NEQ N17:0 N9:40 MOV 18 L203:1 EOR
%   N10:0  SYSTEM_STATE  "STATE The current state of the system" %
%   N9:8  SYSTEM_SUPPLEMENTAL %
%   N17:0  ADS_B_STATE  "STATE The current state of Adsorber B" %
%   N9:40  ADS_STANDBY  "STATE ADS Standby" %
%   L203:1  HMI_STATUS_ADS_B  "HMI Status word for Adsorber B" %

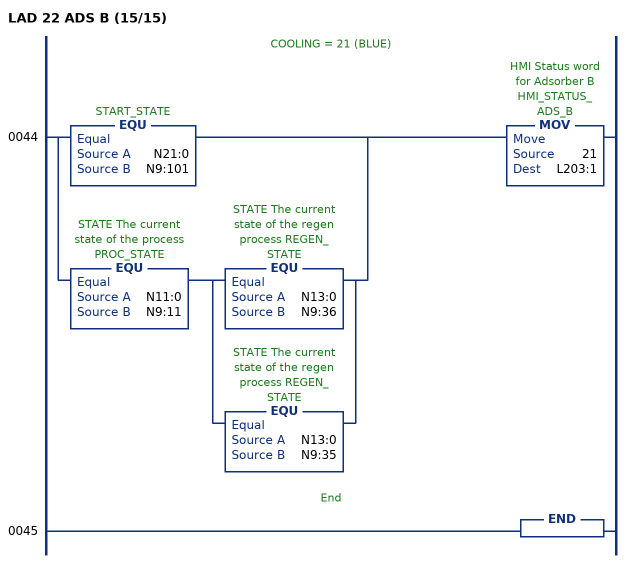
% Rung: 44 %
% COOLING = 21 (BLUE) %
SOR BST EQU N21:0 N9:101 NXB EQU N11:0 N9:11 BST EQU N13:0 N9:36 NXB EQU N13:0 N9:35 BND BND MOV 21 L203:1 EOR
%   N21:0  START_STATE %
%   N9:101  START_COOL %
%   N11:0  PROC_STATE  "STATE The current state of the process" %
%   N9:11  PROC_PFY_A_REG_B  "STATE Process Purify A" %
%   N13:0  REGEN_STATE  "STATE The current state of the regen process" %
%   N9:36  REGEN_COOL  "STATE Regen Cool" %
%   N9:35  REGEN_COOL_WALL  "STATE Regen Cool wall" %
%   L203:1  HMI_STATUS_ADS_B  "HMI Status word for Adsorber B" %
% Rung: 45 %
% End %
SOR END EOR

LADDER 23 "ADS B FLT"    % Controls the Adsorber B faults %
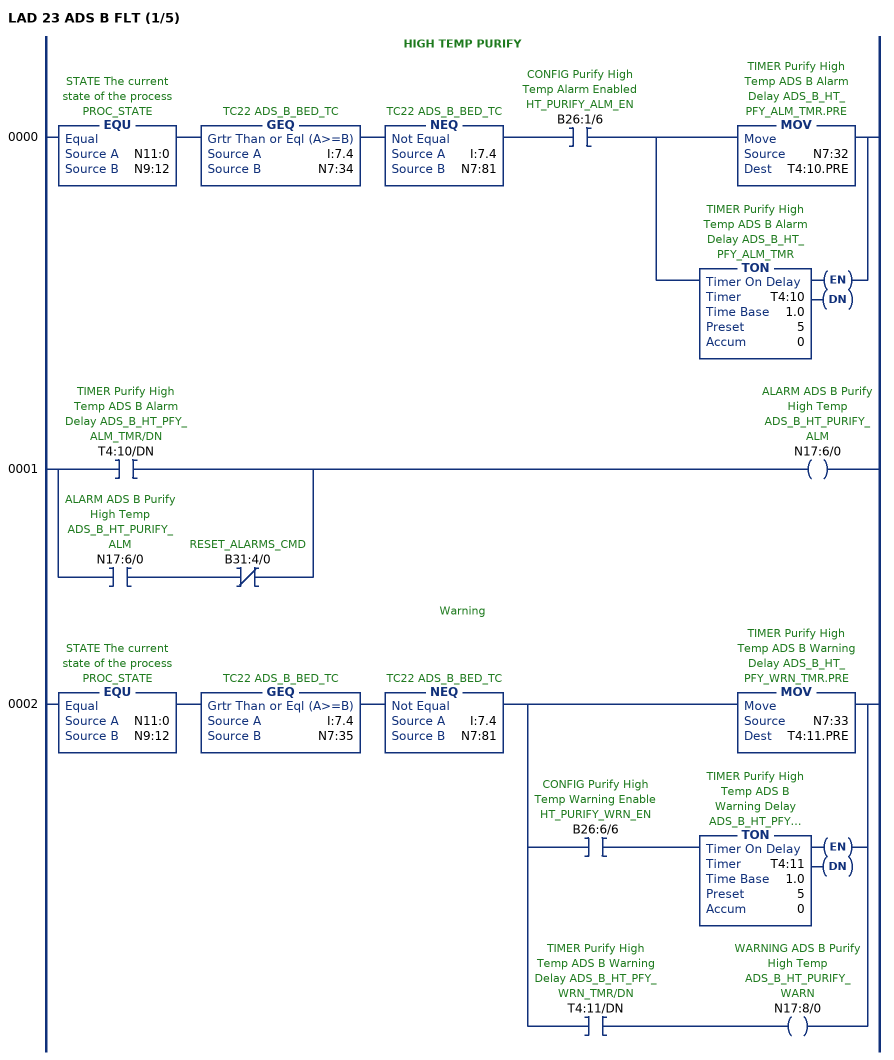
% Rung: 0 %
% TITLE: HIGH TEMP PURIFY %
SOR EQU N11:0 N9:12 GEQ I:7.4 N7:34 NEQ I:7.4 N7:81 XIC B26:1/6 BST MOV N7:32 T4:10.PRE NXB TON T4:10 1.0 5 0 BND EOR
%   N11:0  PROC_STATE  "STATE The current state of the process" %
%   N9:12  PROC_PFY_B_REG_A  "STATE Process Purify B" %
%   I:7.4  ADS_B_BED_TC  "TC22" %
%   N7:34  HT_PURIFY_ALM_SP  "CONFIG Purify High Temp Alarm Setpoint" %
%   N7:81  TC_OPEN_SP  "CONFIG The value read by an open TC input" %
%   B26:1/6  HT_PURIFY_ALM_EN  "CONFIG Purify High Temp Alarm Enabled" %
%   N7:32  HT_PURIFY_ALM_DLY  "CONFIG Purify High Temp Alarm Delay" %
%   T4:10  ADS_B_HT_PFY_ALM_TMR  "TIMER Purify High Temp ADS B Alarm Delay" %
% Rung: 1 %
SOR BST XIC T4:10/DN NXB XIC N17:6/0 XIO B31:4/0 BND OTE N17:6/0 EOR
%   T4:10  ADS_B_HT_PFY_ALM_TMR  "TIMER Purify High Temp ADS B Alarm Delay" %
%   N17:6/0  ADS_B_HT_PURIFY_ALM  "ALARM ADS B Purify High Temp" %
%   B31:4/0  RESET_ALARMS_CMD %
% Rung: 2 %
% Warning %
SOR EQU N11:0 N9:12 GEQ I:7.4 N7:35 NEQ I:7.4 N7:81 BST MOV N7:33 T4:11.PRE NXB XIC B26:6/6 TON T4:11 1.0 5 0 NXB XIC T4:11/DN OTE N17:8/0 BND EOR
%   N11:0  PROC_STATE  "STATE The current state of the process" %
%   N9:12  PROC_PFY_B_REG_A  "STATE Process Purify B" %
%   I:7.4  ADS_B_BED_TC  "TC22" %
%   N7:35  HT_PURIFY_WRN_SP  "CONFIG Purify High Temp Warning Setpoint" %
%   N7:81  TC_OPEN_SP  "CONFIG The value read by an open TC input" %
%   N7:33  HT_PURIFY_WRN_DLY  "CONFIG Purify High Temp Warning Delay" %
%   T4:11  ADS_B_HT_PFY_WRN_TMR  "TIMER Purify High Temp ADS B Warning Delay" %
%   B26:6/6  HT_PURIFY_WRN_EN  "CONFIG Purify High Temp Warning Enable" %
%   N17:8/0  ADS_B_HT_PURIFY_WARN  "WARNING ADS B Purify High Temp" %

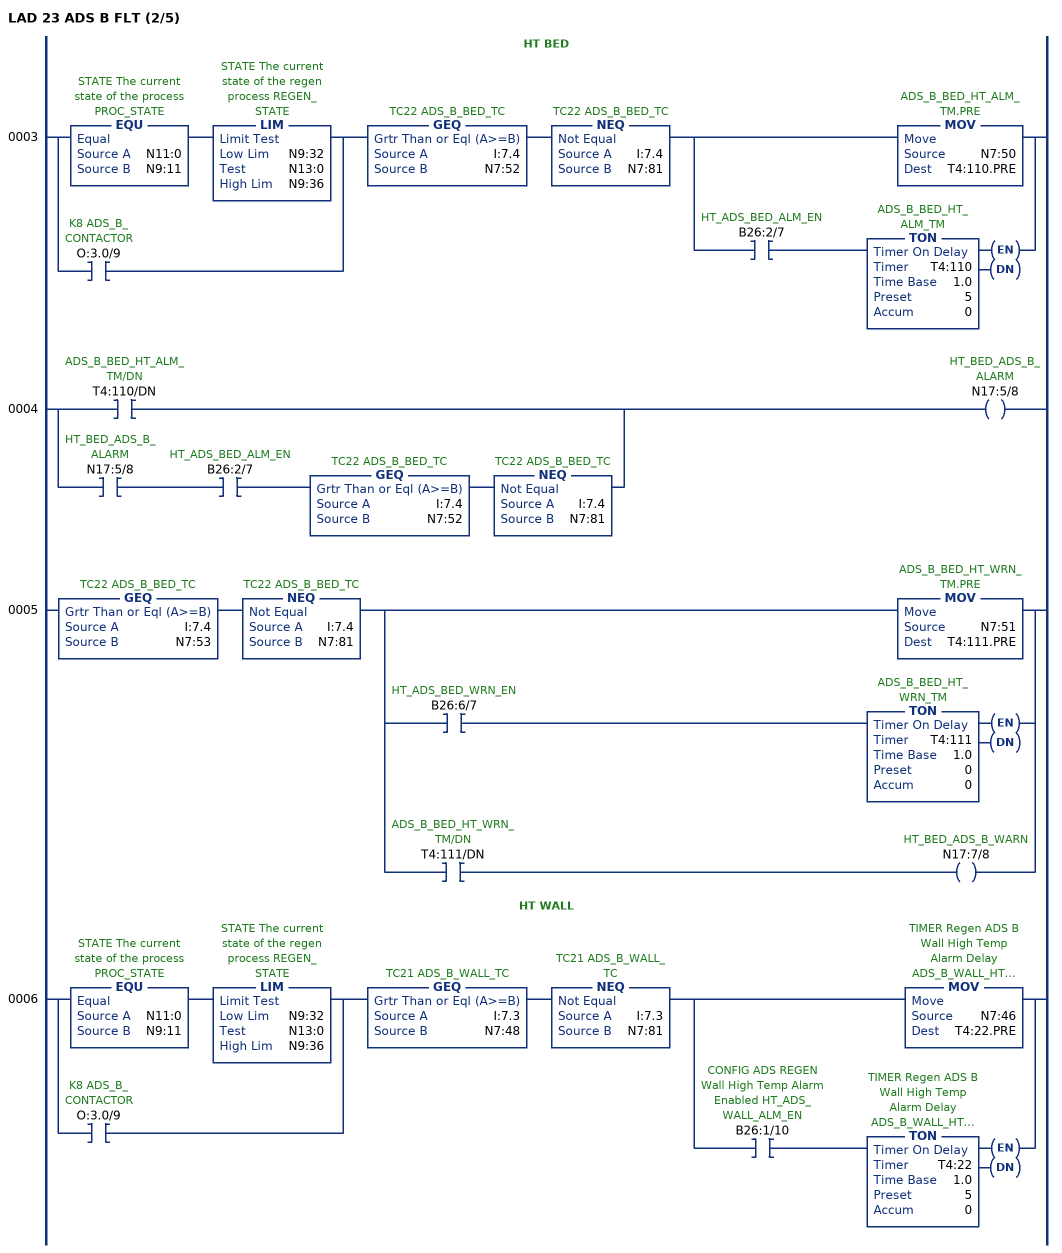
% Rung: 3 %
% TITLE: HT BED %
SOR BST EQU N11:0 N9:11 LIM N9:32 N13:0 N9:36 NXB XIC O:3.0/9 BND GEQ I:7.4 N7:52 NEQ I:7.4 N7:81 BST MOV N7:50 T4:110.PRE NXB XIC B26:2/7 TON T4:110 1.0 5 0 BND EOR
%   N11:0  PROC_STATE  "STATE The current state of the process" %
%   N9:11  PROC_PFY_A_REG_B  "STATE Process Purify A" %
%   N9:32  REGEN_VENT  "STATE Regen Vent" %
%   N13:0  REGEN_STATE  "STATE The current state of the regen process" %
%   N9:36  REGEN_COOL  "STATE Regen Cool" %
%   O:3.0/9  ADS_B_CONTACTOR  "K8" %
%   I:7.4  ADS_B_BED_TC  "TC22" %
%   N7:52  HT_ADS_BED_ALM_SP %
%   N7:81  TC_OPEN_SP  "CONFIG The value read by an open TC input" %
%   N7:50  HT_ADS_BED_ALM_DLY %
%   T4:110  ADS_B_BED_HT_ALM_TM %
%   B26:2/7  HT_ADS_BED_ALM_EN %
% Rung: 4 %
SOR BST XIC T4:110/DN NXB XIC N17:5/8 XIC B26:2/7 GEQ I:7.4 N7:52 NEQ I:7.4 N7:81 BND OTE N17:5/8 EOR
%   T4:110  ADS_B_BED_HT_ALM_TM %
%   N17:5/8  HT_BED_ADS_B_ALARM %
%   B26:2/7  HT_ADS_BED_ALM_EN %
%   I:7.4  ADS_B_BED_TC  "TC22" %
%   N7:52  HT_ADS_BED_ALM_SP %
%   N7:81  TC_OPEN_SP  "CONFIG The value read by an open TC input" %
% Rung: 5 %
SOR GEQ I:7.4 N7:53 NEQ I:7.4 N7:81 BST MOV N7:51 T4:111.PRE NXB XIC B26:6/7 TON T4:111 1.0 0 0 NXB XIC T4:111/DN OTE N17:7/8 BND EOR
%   I:7.4  ADS_B_BED_TC  "TC22" %
%   N7:53  HT_ADS_BED_WRN_SP %
%   N7:81  TC_OPEN_SP  "CONFIG The value read by an open TC input" %
%   N7:51  HT_ADS_BED_WRN_DLY %
%   T4:111  ADS_B_BED_HT_WRN_TM %
%   B26:6/7  HT_ADS_BED_WRN_EN %
%   N17:7/8  HT_BED_ADS_B_WARN %
% Rung: 6 %
% TITLE: HT WALL %
SOR BST EQU N11:0 N9:11 LIM N9:32 N13:0 N9:36 NXB XIC O:3.0/9 BND GEQ I:7.3 N7:48 NEQ I:7.3 N7:81 BST MOV N7:46 T4:22.PRE NXB XIC B26:1/10 TON T4:22 1.0 5 0 BND EOR
%   N11:0  PROC_STATE  "STATE The current state of the process" %
%   N9:11  PROC_PFY_A_REG_B  "STATE Process Purify A" %
%   N9:32  REGEN_VENT  "STATE Regen Vent" %
%   N13:0  REGEN_STATE  "STATE The current state of the regen process" %
%   N9:36  REGEN_COOL  "STATE Regen Cool" %
%   O:3.0/9  ADS_B_CONTACTOR  "K8" %
%   I:7.3  ADS_B_WALL_TC  "TC21" %
%   N7:48  HT_ADS_WALL_ALM_SP  "CONFIG ADS Wall Regen High Temp Alarm" %
%   N7:81  TC_OPEN_SP  "CONFIG The value read by an open TC input" %
%   N7:46  HT_ADS_WALL_ALM_DLY  "CONFIG ADS Wall High Temperature Alarm Delay" %
%   T4:22  ADS_B_WALL_HT_ALM_TM  "TIMER Regen ADS B Wall High Temp Alarm Delay" %
%   B26:1/10  HT_ADS_WALL_ALM_EN  "CONFIG ADS REGEN Wall High Temp Alarm Enabled" %

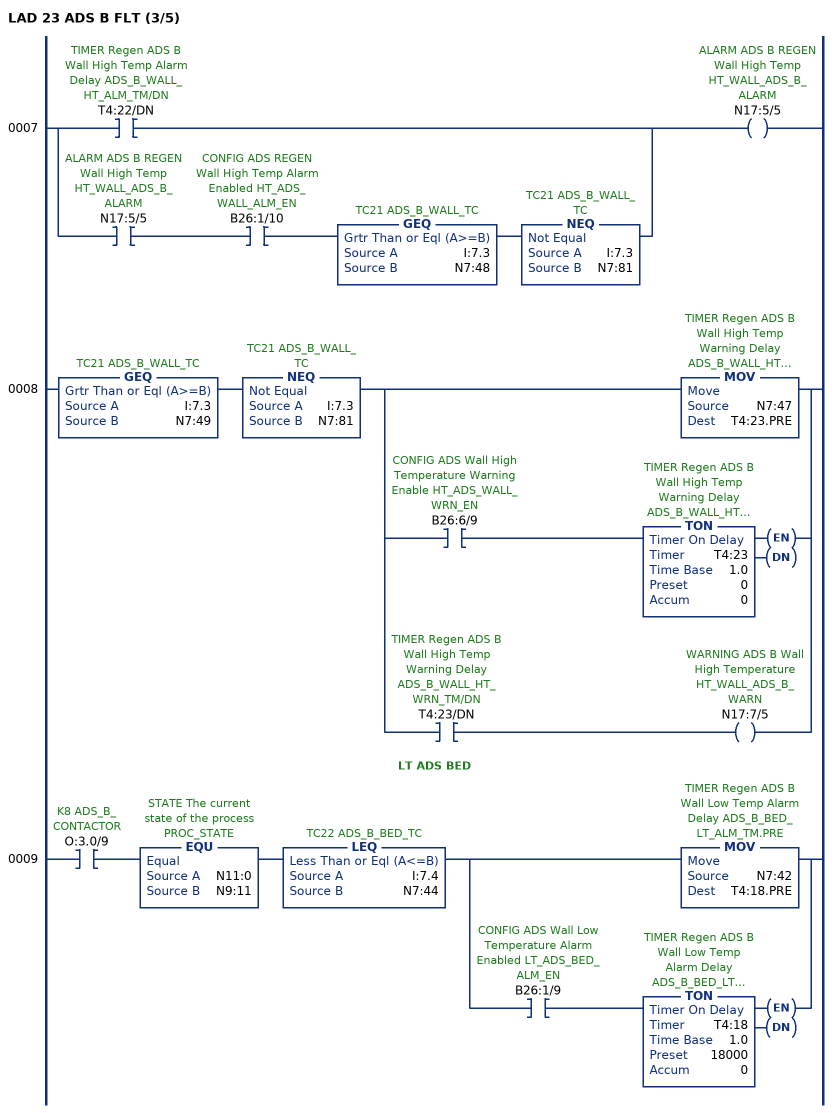
% Rung: 7 %
SOR BST XIC T4:22/DN NXB XIC N17:5/5 XIC B26:1/10 GEQ I:7.3 N7:48 NEQ I:7.3 N7:81 BND OTE N17:5/5 EOR
%   T4:22  ADS_B_WALL_HT_ALM_TM  "TIMER Regen ADS B Wall High Temp Alarm Delay" %
%   N17:5/5  HT_WALL_ADS_B_ALARM  "ALARM ADS B REGEN Wall High Temp" %
%   B26:1/10  HT_ADS_WALL_ALM_EN  "CONFIG ADS REGEN Wall High Temp Alarm Enabled" %
%   I:7.3  ADS_B_WALL_TC  "TC21" %
%   N7:48  HT_ADS_WALL_ALM_SP  "CONFIG ADS Wall Regen High Temp Alarm" %
%   N7:81  TC_OPEN_SP  "CONFIG The value read by an open TC input" %
% Rung: 8 %
SOR GEQ I:7.3 N7:49 NEQ I:7.3 N7:81 BST MOV N7:47 T4:23.PRE NXB XIC B26:6/9 TON T4:23 1.0 0 0 NXB XIC T4:23/DN OTE N17:7/5 BND EOR
%   I:7.3  ADS_B_WALL_TC  "TC21" %
%   N7:49  HT_ADS_WALL_WRN_SP  "CONFIG ADS Wall Regen High Temp Alarm" %
%   N7:81  TC_OPEN_SP  "CONFIG The value read by an open TC input" %
%   N7:47  HT_ADS_WALL_WRN_DLY  "CONFIG ADS Wall High Temperature Warning Delay" %
%   T4:23  ADS_B_WALL_HT_WRN_TM  "TIMER Regen ADS B Wall High Temp Warning Delay" %
%   B26:6/9  HT_ADS_WALL_WRN_EN  "CONFIG ADS Wall High Temperature Warning Enable" %
%   N17:7/5  HT_WALL_ADS_B_WARN  "WARNING ADS B Wall High Temperature" %
% Rung: 9 %
% TITLE: LT ADS BED %
SOR XIC O:3.0/9 EQU N11:0 N9:11 LEQ I:7.4 N7:44 BST MOV N7:42 T4:18.PRE NXB XIC B26:1/9 TON T4:18 1.0 18000 0 BND EOR
%   O:3.0/9  ADS_B_CONTACTOR  "K8" %
%   N11:0  PROC_STATE  "STATE The current state of the process" %
%   N9:11  PROC_PFY_A_REG_B  "STATE Process Purify A" %
%   I:7.4  ADS_B_BED_TC  "TC22" %
%   N7:44  LT_ADS_BED_ALM_SP  "CONFIG ADS Wall Regen Heat Low Temperature Alarm Setpoint" %
%   N7:42  LT_ADS_BED_ALM_DLY  "CONFIG ADS Wall Regen heat Low Temperature Alarm Delay" %
%   T4:18  ADS_B_BED_LT_ALM_TM  "TIMER Regen ADS B Wall Low Temp Alarm Delay" %
%   B26:1/9  LT_ADS_BED_ALM_EN  "CONFIG ADS Wall Low Temperature Alarm Enabled" %

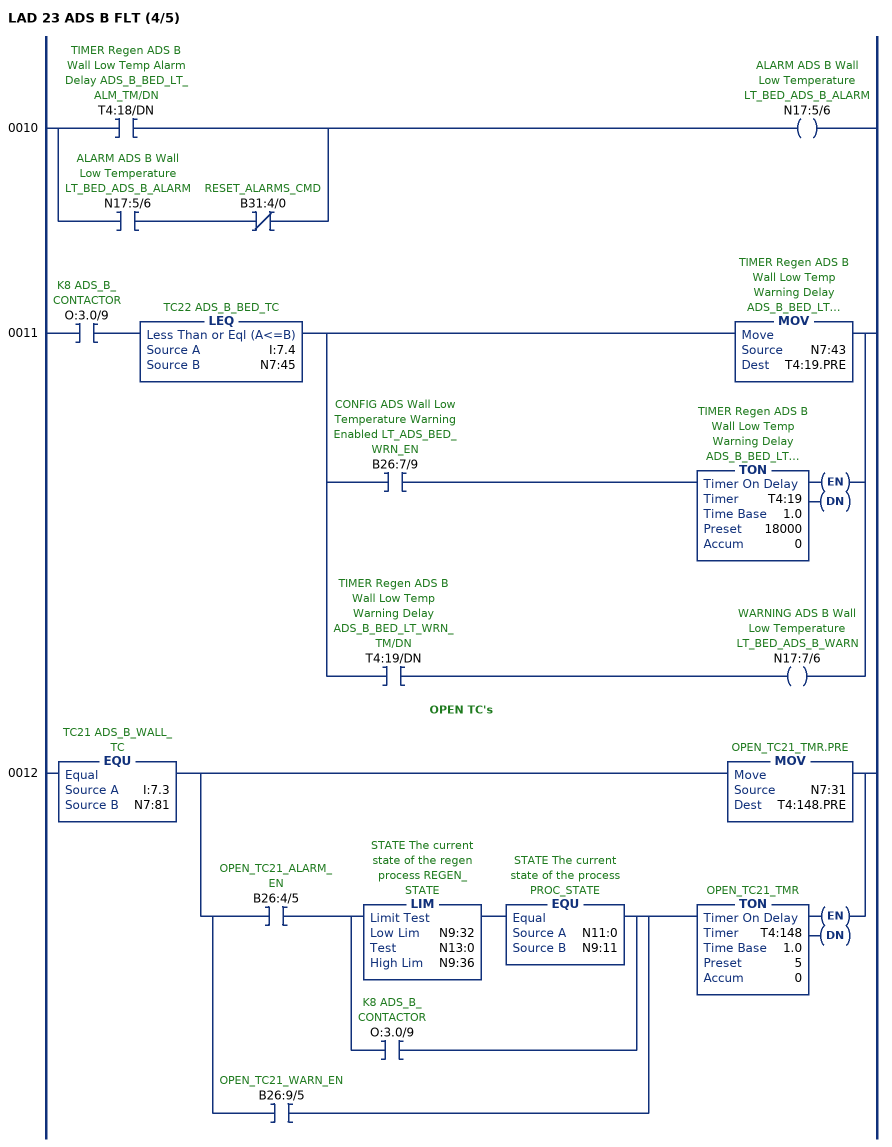
% Rung: 10 %
SOR BST XIC T4:18/DN NXB XIC N17:5/6 XIO B31:4/0 BND OTE N17:5/6 EOR
%   T4:18  ADS_B_BED_LT_ALM_TM  "TIMER Regen ADS B Wall Low Temp Alarm Delay" %
%   N17:5/6  LT_BED_ADS_B_ALARM  "ALARM ADS B Wall Low Temperature" %
%   B31:4/0  RESET_ALARMS_CMD %
% Rung: 11 %
SOR XIC O:3.0/9 LEQ I:7.4 N7:45 BST MOV N7:43 T4:19.PRE NXB XIC B26:7/9 TON T4:19 1.0 18000 0 NXB XIC T4:19/DN OTE N17:7/6 BND EOR
%   O:3.0/9  ADS_B_CONTACTOR  "K8" %
%   I:7.4  ADS_B_BED_TC  "TC22" %
%   N7:45  LT_ADS_BED_WRN_SP  "CONFIG ADS Wall Regen Heat Low Temperature Warning Setpoint" %
%   N7:43  LT_ADS_BED_WRN_DLY  "CONFIG ADS Wall Regen heat Low Temperature Warning Delay" %
%   T4:19  ADS_B_BED_LT_WRN_TM  "TIMER Regen ADS B Wall Low Temp Warning Delay" %
%   B26:7/9  LT_ADS_BED_WRN_EN  "CONFIG ADS Wall Low Temperature Warning Enabled" %
%   N17:7/6  LT_BED_ADS_B_WARN  "WARNING ADS B Wall Low Temperature" %
% Rung: 12 %
% TITLE: OPEN TC's %
SOR EQU I:7.3 N7:81 BST MOV N7:31 T4:148.PRE NXB BST XIC B26:4/5 BST LIM N9:32 N13:0 N9:36 EQU N11:0 N9:11 NXB XIC O:3.0/9 BND NXB XIC B26:9/5 BND TON T4:148 1.0 5 0 BND EOR
%   I:7.3  ADS_B_WALL_TC  "TC21" %
%   N7:81  TC_OPEN_SP  "CONFIG The value read by an open TC input" %
%   N7:31  OPEN_TC_DLY %
%   T4:148  OPEN_TC21_TMR %
%   B26:4/5  OPEN_TC21_ALARM_EN %
%   N9:32  REGEN_VENT  "STATE Regen Vent" %
%   N13:0  REGEN_STATE  "STATE The current state of the regen process" %
%   N9:36  REGEN_COOL  "STATE Regen Cool" %
%   N11:0  PROC_STATE  "STATE The current state of the process" %
%   N9:11  PROC_PFY_A_REG_B  "STATE Process Purify A" %
%   O:3.0/9  ADS_B_CONTACTOR  "K8" %
%   B26:9/5  OPEN_TC21_WARN_EN %

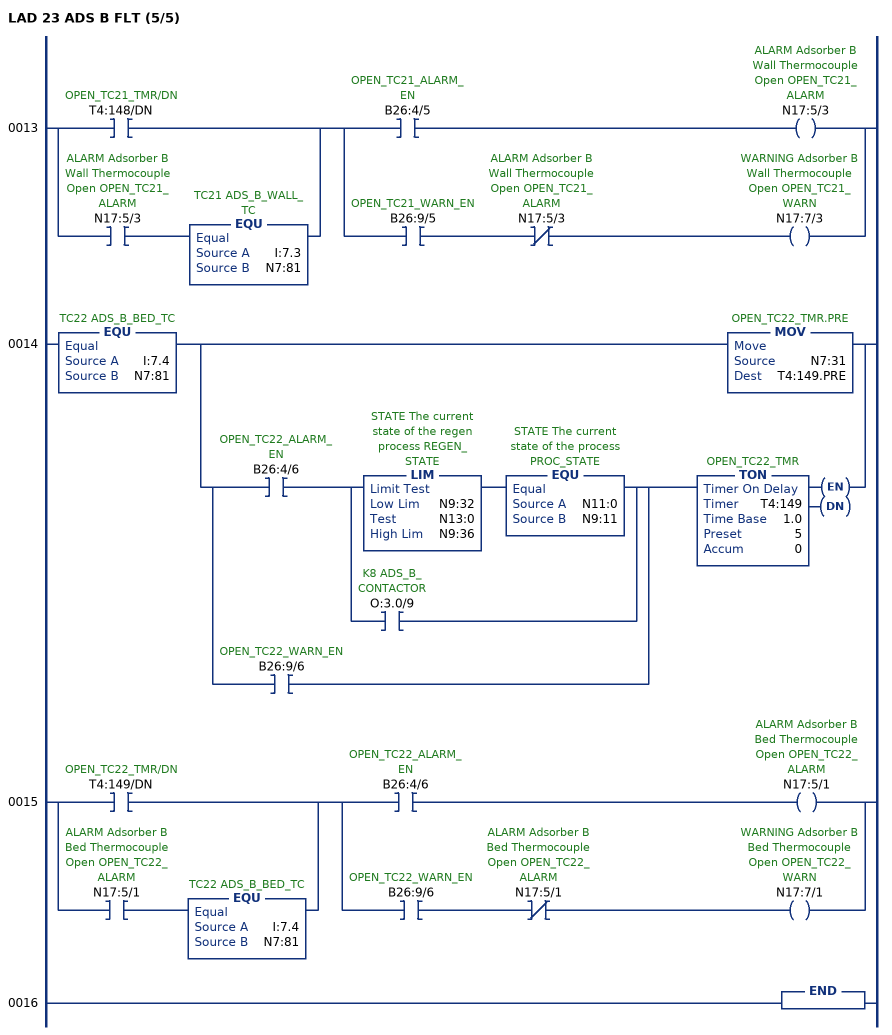
% Rung: 13 %
SOR BST XIC T4:148/DN NXB XIC N17:5/3 EQU I:7.3 N7:81 BND BST XIC B26:4/5 OTE N17:5/3 NXB XIC B26:9/5 XIO N17:5/3 OTE N17:7/3 BND EOR
%   T4:148  OPEN_TC21_TMR %
%   N17:5/3  OPEN_TC21_ALARM  "ALARM Adsorber B Wall Thermocouple Open" %
%   I:7.3  ADS_B_WALL_TC  "TC21" %
%   N7:81  TC_OPEN_SP  "CONFIG The value read by an open TC input" %
%   B26:4/5  OPEN_TC21_ALARM_EN %
%   B26:9/5  OPEN_TC21_WARN_EN %
%   N17:7/3  OPEN_TC21_WARN  "WARNING Adsorber B Wall Thermocouple Open" %
% Rung: 14 %
SOR EQU I:7.4 N7:81 BST MOV N7:31 T4:149.PRE NXB BST XIC B26:4/6 BST LIM N9:32 N13:0 N9:36 EQU N11:0 N9:11 NXB XIC O:3.0/9 BND NXB XIC B26:9/6 BND TON T4:149 1.0 5 0 BND EOR
%   I:7.4  ADS_B_BED_TC  "TC22" %
%   N7:81  TC_OPEN_SP  "CONFIG The value read by an open TC input" %
%   N7:31  OPEN_TC_DLY %
%   T4:149  OPEN_TC22_TMR %
%   B26:4/6  OPEN_TC22_ALARM_EN %
%   N9:32  REGEN_VENT  "STATE Regen Vent" %
%   N13:0  REGEN_STATE  "STATE The current state of the regen process" %
%   N9:36  REGEN_COOL  "STATE Regen Cool" %
%   N11:0  PROC_STATE  "STATE The current state of the process" %
%   N9:11  PROC_PFY_A_REG_B  "STATE Process Purify A" %
%   O:3.0/9  ADS_B_CONTACTOR  "K8" %
%   B26:9/6  OPEN_TC22_WARN_EN %
% Rung: 15 %
SOR BST XIC T4:149/DN NXB XIC N17:5/1 EQU I:7.4 N7:81 BND BST XIC B26:4/6 OTE N17:5/1 NXB XIC B26:9/6 XIO N17:5/1 OTE N17:7/1 BND EOR
%   T4:149  OPEN_TC22_TMR %
%   N17:5/1  OPEN_TC22_ALARM  "ALARM Adsorber B Bed Thermocouple Open" %
%   I:7.4  ADS_B_BED_TC  "TC22" %
%   N7:81  TC_OPEN_SP  "CONFIG The value read by an open TC input" %
%   B26:4/6  OPEN_TC22_ALARM_EN %
%   B26:9/6  OPEN_TC22_WARN_EN %
%   N17:7/1  OPEN_TC22_WARN  "WARNING Adsorber B Bed Thermocouple Open" %
% Rung: 16 %
SOR END EOR

LADDER 24 "ADS PH"
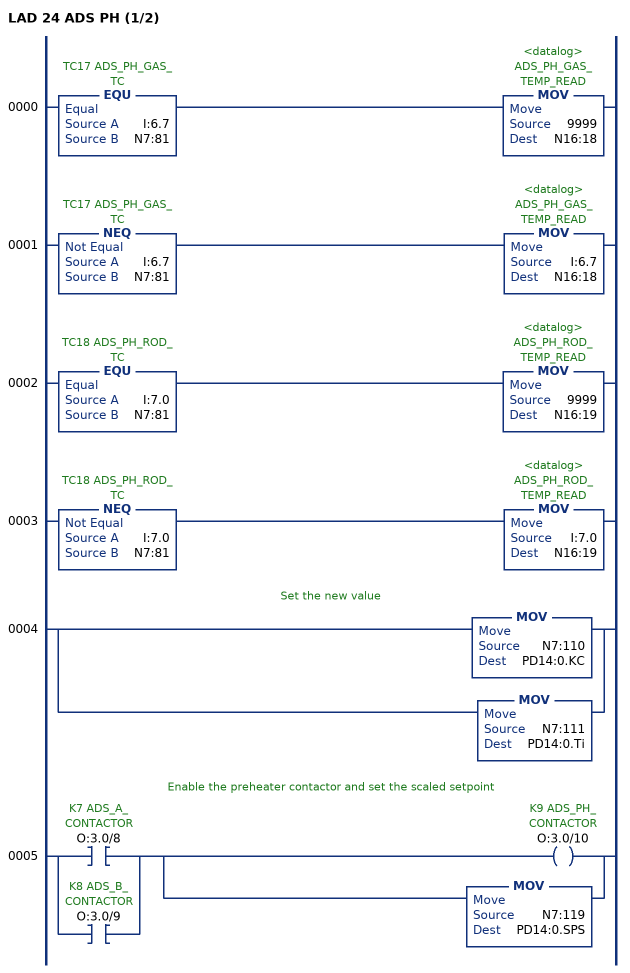
% Rung: 0 %
SOR EQU I:6.7 N7:81 MOV 9999 N16:18 EOR
%   I:6.7  ADS_PH_GAS_TC  "TC17" %
%   N7:81  TC_OPEN_SP  "CONFIG The value read by an open TC input" %
%   N16:18  ADS_PH_GAS_TEMP_READ  "<datalog>" %
% Rung: 1 %
SOR NEQ I:6.7 N7:81 MOV I:6.7 N16:18 EOR
%   I:6.7  ADS_PH_GAS_TC  "TC17" %
%   N7:81  TC_OPEN_SP  "CONFIG The value read by an open TC input" %
%   N16:18  ADS_PH_GAS_TEMP_READ  "<datalog>" %
% Rung: 2 %
SOR EQU I:7.0 N7:81 MOV 9999 N16:19 EOR
%   I:7.0  ADS_PH_ROD_TC  "TC18" %
%   N7:81  TC_OPEN_SP  "CONFIG The value read by an open TC input" %
%   N16:19  ADS_PH_ROD_TEMP_READ  "<datalog>" %
% Rung: 3 %
SOR NEQ I:7.0 N7:81 MOV I:7.0 N16:19 EOR
%   I:7.0  ADS_PH_ROD_TC  "TC18" %
%   N7:81  TC_OPEN_SP  "CONFIG The value read by an open TC input" %
%   N16:19  ADS_PH_ROD_TEMP_READ  "<datalog>" %
% Rung: 4 %
% Set the new value %
SOR BST MOV N7:110 PD14:0.KC NXB MOV N7:111 PD14:0.Ti BND EOR
%   N7:110  PREHEATER_P  "CONFIG Preheater Proportional Gain New" %
%   N7:111  PREHEATER_I  "CONFIG Preheater Integral Gain New" %
% Rung: 5 %
% Enable the preheater contactor and set the scaled setpoint %
SOR BST XIC O:3.0/8 NXB XIC O:3.0/9 BND BST OTE O:3.0/10 NXB MOV N7:119 PD14:0.SPS BND EOR
%   O:3.0/8  ADS_A_CONTACTOR  "K7" %
%   O:3.0/9  ADS_B_CONTACTOR  "K8" %
%   O:3.0/10  ADS_PH_CONTACTOR  "K9" %
%   N7:119  PREHEATER_SP  "<datalog> CONTROL Preheater PID Setpoint" %

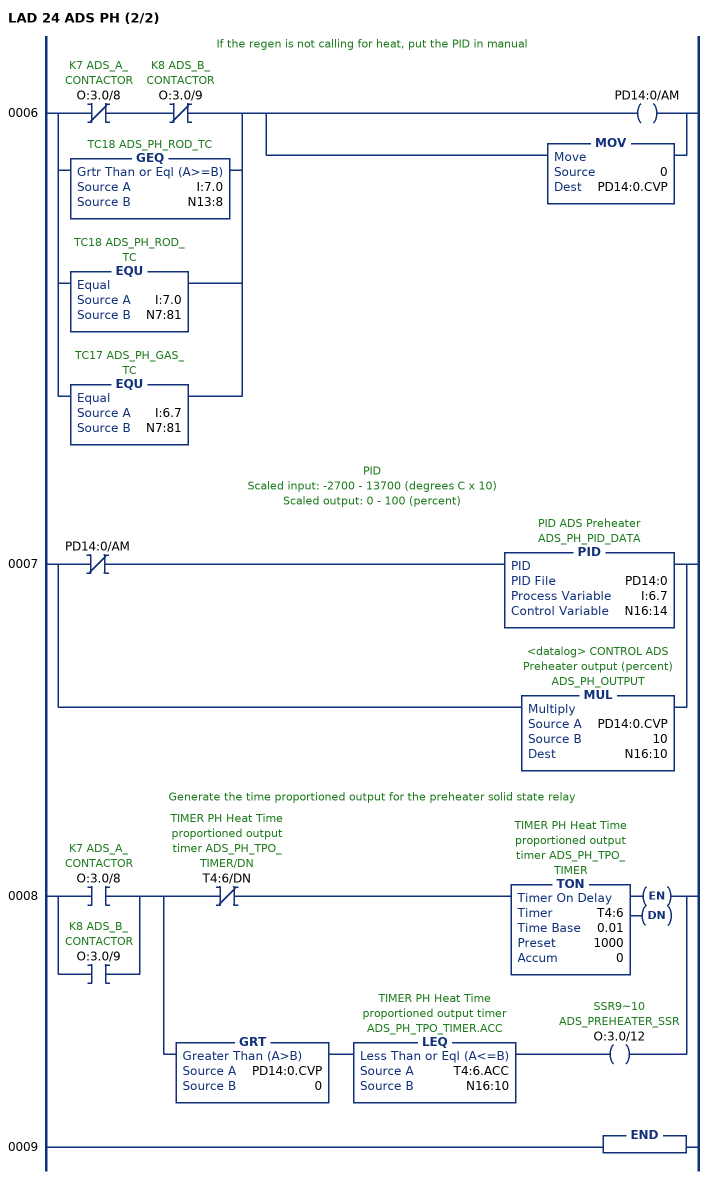
% Rung: 6 %
% If the regen is not calling for heat, put the PID in manual %
SOR BST XIO O:3.0/8 XIO O:3.0/9 NXB GEQ I:7.0 N13:8 NXB EQU I:7.0 N7:81 NXB EQU I:6.7 N7:81 BND BST OTE PD14:0/AM NXB MOV 0 PD14:0.CVP BND EOR
%   O:3.0/8  ADS_A_CONTACTOR  "K7" %
%   O:3.0/9  ADS_B_CONTACTOR  "K8" %
%   I:7.0  ADS_PH_ROD_TC  "TC18" %
%   N13:8  PH_ROD_LIMIT %
%   N7:81  TC_OPEN_SP  "CONFIG The value read by an open TC input" %
%   I:6.7  ADS_PH_GAS_TC  "TC17" %
% Rung: 7 %
% PID
% Scaled input: -2700 - 13700 (degrees C x 10)
% Scaled output: 0 - 100 (percent) %
SOR BST XIO PD14:0/AM PID PD14:0 I:6.7 N16:14 NXB MUL PD14:0.CVP 10 N16:10 BND EOR
%   PD14:0  ADS_PH_PID_DATA  "PID ADS Preheater" %
%   I:6.7  ADS_PH_GAS_TC  "TC17" %
%   N16:14  ADS_PH_OUTPUT_RAW  "CONTROL ADS A Preheater PID Output Raw" %
%   N16:10  ADS_PH_OUTPUT  "<datalog> CONTROL ADS Preheater output (percent)" %
% Rung: 8 %
% Generate the time proportioned output for the preheater solid state relay %
SOR BST XIC O:3.0/8 NXB XIC O:3.0/9 BND BST XIO T4:6/DN TON T4:6 0.01 1000 0 NXB GRT PD14:0.CVP 0 LEQ T4:6.ACC N16:10 OTE O:3.0/12 BND EOR
%   O:3.0/8  ADS_A_CONTACTOR  "K7" %
%   O:3.0/9  ADS_B_CONTACTOR  "K8" %
%   T4:6  ADS_PH_TPO_TIMER  "TIMER PH Heat Time proportioned output timer" %
%   N16:10  ADS_PH_OUTPUT  "<datalog> CONTROL ADS Preheater output (percent)" %
%   O:3.0/12  ADS_PREHEATER_SSR  "SSR9~10" %
% Rung: 9 %
SOR END EOR

LADDER 25 "ADS PH FLT"
